   DATA[1204,17] := 1.0;
   DATA[1204,18] := 1.0;
   DATA[1204,19] := 1.0;
   DATA[1204,20] := 148.808;
   DATA[1204,21] := 154.2425;
   DATA[1204,22] := 1.716721;
   DATA[1204,23] := 841.2843;
   DATA[1204,24] := 2.0;
   DATA[1204,25] := 2.0;
   DATA[1204,26] := 7.87798;
   DATA[1204,27] := 143.5786;
   DATA[1204,28] := 263.0095;
   DATA[1204,29] := 12.07383;
   DATA[1204,30] := 1.725968;
   DATA[1204,31] := 1.298578;
   DATA[1204,32] := 0.7352687;
   DATA[1204,33] := 0.3083624;
   DATA[1204,34] := 2.0;
   DATA[1204,35] := 250.4166;
   DATA[1204,36] := 1.69801;
   DATA[1204,37] := 189.2944;
   DATA[1204,38] := 0.000128152;
   DATA[1204,39] := 1.0;
   DATA[1205,0] := 2.554527;
   DATA[1205,1] := 754.2025;
   DATA[1205,2] := 2.0;
   DATA[1205,3] := 1.0;
   DATA[1205,4] := 262.5288;
   DATA[1205,5] := 8.464369;
   DATA[1205,6] := 317.1494;
   DATA[1205,8] := 1.0;
   DATA[1205,9] := 1.0;
   DATA[1205,10] := 1.0;
   DATA[1205,11] := 2.010372;
   DATA[1205,12] := 0.000256221;
   DATA[1205,13] := 1011.079;
   DATA[1205,14] := 1.0;
   DATA[1205,15] := 1.0;
   DATA[1205,16] := 1.0;
   DATA[1205,17] := 1.0;
   DATA[1205,18] := 1.0;
   DATA[1205,19] := 1.0;
   DATA[1205,20] := 148.808;
   DATA[1205,21] := 154.2425;
   DATA[1205,22] := 1.717233;
   DATA[1205,23] := 840.8998;
   DATA[1205,24] := 2.0;
   DATA[1205,25] := 2.0;
   DATA[1205,26] := 7.87798;
   DATA[1205,27] := 143.5786;
   DATA[1205,28] := 263.0095;
   DATA[1205,29] := 12.26609;
   DATA[1205,30] := 1.725968;
   DATA[1205,31] := 1.301396;
   DATA[1205,32] := 0.7352687;
   DATA[1205,33] := 0.3083624;
   DATA[1205,34] := 2.0;
   DATA[1205,35] := 250.2724;
   DATA[1205,36] := 1.69801;
   DATA[1205,37] := 189.1342;
   DATA[1205,38] := 0.000128152;
   DATA[1205,39] := 1.0;
   DATA[1206,0] := 2.554527;
   DATA[1206,1] := 754.7128;
   DATA[1206,2] := 2.0;
   DATA[1206,3] := 1.0;
   DATA[1206,4] := 262.5288;
   DATA[1206,5] := 8.464369;
   DATA[1206,6] := 317.1494;
   DATA[1206,8] := 1.0;
   DATA[1206,9] := 1.0;
   DATA[1206,10] := 1.0;
   DATA[1206,11] := 2.010372;
   DATA[1206,12] := 0.000256221;
   DATA[1206,13] := 1010.919;
   DATA[1206,14] := 1.0;
   DATA[1206,15] := 1.0;
   DATA[1206,16] := 1.0;
   DATA[1206,17] := 1.0;
   DATA[1206,18] := 1.0;
   DATA[1206,19] := 1.0;
   DATA[1206,20] := 148.808;
   DATA[1206,21] := 154.2425;
   DATA[1206,22] := 1.717874;
   DATA[1206,23] := 840.7844;
   DATA[1206,24] := 2.0;
   DATA[1206,25] := 2.0;
   DATA[1206,26] := 7.87798;
   DATA[1206,27] := 143.5786;
   DATA[1206,28] := 263.0095;
   DATA[1206,29] := 12.26609;
   DATA[1206,30] := 1.72443;
   DATA[1206,31] := 1.291789;
   DATA[1206,32] := 0.7352687;
   DATA[1206,33] := 0.3083624;
   DATA[1206,34] := 2.0;
   DATA[1206,35] := 250.2724;
   DATA[1206,36] := 1.69801;
   DATA[1206,37] := 189.0381;
   DATA[1206,38] := 0.000128152;
   DATA[1206,39] := 1.0;
   DATA[1207,0] := 2.554527;
   DATA[1207,1] := 755.2623;
   DATA[1207,2] := 2.0;
   DATA[1207,3] := 1.0;
   DATA[1207,4] := 262.5288;
   DATA[1207,5] := 8.464369;
   DATA[1207,6] := 317.1494;
   DATA[1207,8] := 1.0;
   DATA[1207,9] := 1.0;
   DATA[1207,10] := 1.0;
   DATA[1207,11] := 2.010372;
   DATA[1207,12] := 0.000256221;
   DATA[1207,13] := 1011.159;
   DATA[1207,14] := 1.0;
   DATA[1207,15] := 1.0;
   DATA[1207,16] := 1.0;
   DATA[1207,17] := 1.0;
   DATA[1207,18] := 1.0;
   DATA[1207,19] := 1.0;
   DATA[1207,20] := 148.808;
   DATA[1207,21] := 154.2425;
   DATA[1207,22] := 1.717874;
   DATA[1207,23] := 840.2845;
   DATA[1207,24] := 2.0;
   DATA[1207,25] := 2.0;
   DATA[1207,26] := 7.87798;
   DATA[1207,27] := 143.4248;
   DATA[1207,28] := 263.0095;
   DATA[1207,29] := 12.26609;
   DATA[1207,30] := 1.722892;
   DATA[1207,31] := 1.284232;
   DATA[1207,32] := 0.7352687;
   DATA[1207,33] := 0.3083624;
   DATA[1207,34] := 2.0;
   DATA[1207,35] := 250.1442;
   DATA[1207,36] := 1.69801;
   DATA[1207,37] := 189.0381;
   DATA[1207,38] := 0.000128152;
   DATA[1207,39] := 1.0;
   DATA[1208,0] := 2.55805;
   DATA[1208,1] := 755.6941;
   DATA[1208,2] := 2.0;
   DATA[1208,3] := 1.0;
   DATA[1208,4] := 262.5288;
   DATA[1208,5] := 8.464369;
   DATA[1208,6] := 317.1494;
   DATA[1208,8] := 1.0;
   DATA[1208,9] := 1.0;
   DATA[1208,10] := 1.0;
   DATA[1208,11] := 2.010372;
   DATA[1208,12] := 0.000256221;
   DATA[1208,13] := 1010.718;
   DATA[1208,14] := 1.0;
   DATA[1208,15] := 1.0;
   DATA[1208,16] := 1.0;
   DATA[1208,17] := 1.0;
   DATA[1208,18] := 1.0;
   DATA[1208,19] := 1.0;
   DATA[1208,20] := 148.808;
   DATA[1208,21] := 154.2425;
   DATA[1208,22] := 1.717874;
   DATA[1208,23] := 840.2076;
   DATA[1208,24] := 2.0;
   DATA[1208,25] := 2.0;
   DATA[1208,26] := 7.87798;
   DATA[1208,27] := 143.4248;
   DATA[1208,28] := 263.0095;
   DATA[1208,29] := 12.03538;
   DATA[1208,30] := 1.722892;
   DATA[1208,31] := 1.272576;
   DATA[1208,32] := 0.7352687;
   DATA[1208,33] := 0.3083624;
   DATA[1208,34] := 2.0;
   DATA[1208,35] := 250.1442;
   DATA[1208,36] := 1.69801;
   DATA[1208,37] := 189.0381;
   DATA[1208,38] := 0.000128152;
   DATA[1208,39] := 1.0;
   DATA[1209,0] := 2.559651;
   DATA[1209,1] := 756.4791;
   DATA[1209,2] := 2.0;
   DATA[1209,3] := 1.0;
   DATA[1209,4] := 262.5288;
   DATA[1209,5] := 8.464369;
   DATA[1209,6] := 317.1494;
   DATA[1209,8] := 1.0;
   DATA[1209,9] := 1.0;
   DATA[1209,10] := 1.0;
   DATA[1209,11] := 2.010372;
   DATA[1209,12] := 0.000256221;
   DATA[1209,13] := 1010.919;
   DATA[1209,14] := 1.0;
   DATA[1209,15] := 1.0;
   DATA[1209,16] := 1.0;
   DATA[1209,17] := 1.0;
   DATA[1209,18] := 1.0;
   DATA[1209,19] := 1.0;
   DATA[1209,20] := 148.808;
   DATA[1209,21] := 154.1912;
   DATA[1209,22] := 1.715439;
   DATA[1209,23] := 839.9;
   DATA[1209,24] := 2.0;
   DATA[1209,25] := 2.0;
   DATA[1209,26] := 7.87798;
   DATA[1209,27] := 143.4248;
   DATA[1209,28] := 263.0095;
   DATA[1209,29] := 12.03538;
   DATA[1209,30] := 1.722892;
   DATA[1209,31] := 1.263738;
   DATA[1209,32] := 0.7352687;
   DATA[1209,33] := 0.3083624;
   DATA[1209,34] := 2.0;
   DATA[1209,35] := 250.1442;
   DATA[1209,36] := 1.69801;
   DATA[1209,37] := 189.0381;
   DATA[1209,38] := 0.000128152;
   DATA[1209,39] := 1.0;
   DATA[1210,0] := 2.550043;
   DATA[1210,1] := 756.9502;
   DATA[1210,2] := 2.0;
   DATA[1210,3] := 1.0;
   DATA[1210,4] := 262.5288;
   DATA[1210,5] := 8.464369;
   DATA[1210,6] := 317.1494;
   DATA[1210,8] := 1.0;
   DATA[1210,9] := 1.0;
   DATA[1210,10] := 1.0;
   DATA[1210,11] := 2.010372;
   DATA[1210,12] := 0.000256221;
   DATA[1210,13] := 1010.879;
   DATA[1210,14] := 1.0;
   DATA[1210,15] := 1.0;
   DATA[1210,16] := 1.0;
   DATA[1210,17] := 1.0;
   DATA[1210,18] := 1.0;
   DATA[1210,19] := 1.0;
   DATA[1210,20] := 148.808;
   DATA[1210,21] := 154.0374;
   DATA[1210,22] := 1.713261;
   DATA[1210,23] := 839.2848;
   DATA[1210,24] := 2.0;
   DATA[1210,25] := 2.0;
   DATA[1210,26] := 7.87798;
   DATA[1210,27] := 143.4248;
   DATA[1210,28] := 263.0095;
   DATA[1210,29] := 12.03538;
   DATA[1210,30] := 1.722892;
   DATA[1210,31] := 1.279237;
   DATA[1210,32] := 0.7352687;
   DATA[1210,33] := 0.3083624;
   DATA[1210,34] := 2.0;
   DATA[1210,35] := 250.1442;
   DATA[1210,36] := 1.69801;
   DATA[1210,37] := 189.0381;
   DATA[1210,38] := 0.000128152;
   DATA[1210,39] := 1.0;
   DATA[1211,0] := 2.550043;
   DATA[1211,1] := 757.853;
   DATA[1211,2] := 2.0;
   DATA[1211,3] := 1.0;
   DATA[1211,4] := 262.5288;
   DATA[1211,5] := 8.464369;
   DATA[1211,6] := 317.1494;
   DATA[1211,8] := 1.0;
   DATA[1211,9] := 1.0;
   DATA[1211,10] := 1.0;
   DATA[1211,11] := 2.010372;
   DATA[1211,12] := 0.000256221;
   DATA[1211,13] := 1010.879;
   DATA[1211,14] := 1.0;
   DATA[1211,15] := 1.0;
   DATA[1211,16] := 1.0;
   DATA[1211,17] := 1.0;
   DATA[1211,18] := 1.0;
   DATA[1211,19] := 1.0;
   DATA[1211,20] := 148.808;
   DATA[1211,21] := 153.8836;
   DATA[1211,22] := 1.711723;
   DATA[1211,23] := 839.3232;
   DATA[1211,24] := 2.0;
   DATA[1211,25] := 2.0;
   DATA[1211,26] := 7.87798;
   DATA[1211,27] := 143.4248;
   DATA[1211,28] := 263.0095;
   DATA[1211,29] := 12.03538;
   DATA[1211,30] := 1.722379;
   DATA[1211,31] := 1.289484;
   DATA[1211,32] := 0.7352687;
   DATA[1211,33] := 0.3083624;
   DATA[1211,34] := 2.0;
   DATA[1211,35] := 250.1442;
   DATA[1211,36] := 1.69801;
   DATA[1211,37] := 189.0381;
   DATA[1211,38] := 0.000128152;
   DATA[1211,39] := 1.0;
   DATA[1212,0] := 2.552285;
   DATA[1212,1] := 758.0885;
   DATA[1212,2] := 2.0;
   DATA[1212,3] := 1.0;
   DATA[1212,4] := 262.5288;
   DATA[1212,5] := 8.464369;
   DATA[1212,6] := 317.1494;
   DATA[1212,8] := 1.0;
   DATA[1212,9] := 1.0;
   DATA[1212,10] := 1.0;
   DATA[1212,11] := 2.010372;
   DATA[1212,12] := 0.000256221;
   DATA[1212,13] := 1010.718;
   DATA[1212,14] := 1.0;
   DATA[1212,15] := 1.0;
   DATA[1212,16] := 1.0;
   DATA[1212,17] := 1.0;
   DATA[1212,18] := 1.0;
   DATA[1212,19] := 1.0;
   DATA[1212,20] := 148.808;
   DATA[1212,21] := 153.8836;
   DATA[1212,22] := 1.711082;
   DATA[1212,23] := 838.8618;
   DATA[1212,24] := 2.0;
   DATA[1212,25] := 2.0;
   DATA[1212,26] := 7.87798;
   DATA[1212,27] := 143.4248;
   DATA[1212,28] := 263.0095;
   DATA[1212,29] := 12.03538;
   DATA[1212,30] := 1.722379;
   DATA[1212,31] := 1.299731;
   DATA[1212,32] := 0.7352687;
   DATA[1212,33] := 0.3083624;
   DATA[1212,34] := 2.0;
   DATA[1212,35] := 250.3525;
   DATA[1212,36] := 1.69801;
   DATA[1212,37] := 189.0381;
   DATA[1212,38] := 0.000128152;
   DATA[1212,39] := 1.0;
   DATA[1213,0] := 2.554847;
   DATA[1213,1] := 758.7166;
   DATA[1213,2] := 2.0;
   DATA[1213,3] := 1.0;
   DATA[1213,4] := 262.5288;
   DATA[1213,5] := 8.464369;
   DATA[1213,6] := 317.1494;
   DATA[1213,8] := 1.0;
   DATA[1213,9] := 1.0;
   DATA[1213,10] := 1.0;
   DATA[1213,11] := 2.010372;
   DATA[1213,12] := 0.000256221;
   DATA[1213,13] := 1010.478;
   DATA[1213,14] := 1.0;
   DATA[1213,15] := 1.0;
   DATA[1213,16] := 1.0;
   DATA[1213,17] := 1.0;
   DATA[1213,18] := 1.0;
   DATA[1213,19] := 1.0;
   DATA[1213,20] := 148.808;
   DATA[1213,21] := 153.8836;
   DATA[1213,22] := 1.711082;
   DATA[1213,23] := 838.5542;
   DATA[1213,24] := 2.0;
   DATA[1213,25] := 2.0;
   DATA[1213,26] := 7.87798;
   DATA[1213,27] := 143.4248;
   DATA[1213,28] := 263.0095;
   DATA[1213,29] := 12.03538;
   DATA[1213,30] := 1.722379;
   DATA[1213,31] := 1.30114;
   DATA[1213,32] := 0.7352687;
   DATA[1213,33] := 0.3083624;
   DATA[1213,34] := 2.0;
   DATA[1213,35] := 250.3525;
   DATA[1213,36] := 1.69801;
   DATA[1213,37] := 189.0541;
   DATA[1213,38] := 0.000128152;
   DATA[1213,39] := 1.0;
   DATA[1214,0] := 2.556129;
   DATA[1214,1] := 759.4231;
   DATA[1214,2] := 2.0;
   DATA[1214,3] := 1.0;
   DATA[1214,4] := 262.5288;
   DATA[1214,5] := 8.464369;
   DATA[1214,6] := 317.1494;
   DATA[1214,8] := 1.0;
   DATA[1214,9] := 1.0;
   DATA[1214,10] := 1.0;
   DATA[1214,11] := 2.010372;
   DATA[1214,12] := 0.000256221;
   DATA[1214,13] := 1010.718;
   DATA[1214,14] := 1.0;
   DATA[1214,15] := 1.0;
   DATA[1214,16] := 1.0;
   DATA[1214,17] := 1.0;
   DATA[1214,18] := 1.0;
   DATA[1214,19] := 1.0;
   DATA[1214,20] := 148.808;
   DATA[1214,21] := 154.0118;
   DATA[1214,22] := 1.712363;
   DATA[1214,23] := 838.0543;
   DATA[1214,24] := 2.0;
   DATA[1214,25] := 2.0;
   DATA[1214,26] := 7.87798;
   DATA[1214,27] := 143.3222;
   DATA[1214,28] := 263.0095;
   DATA[1214,29] := 12.03538;
   DATA[1214,30] := 1.725583;
   DATA[1214,31] := 1.291789;
   DATA[1214,32] := 0.7352687;
   DATA[1214,33] := 0.3074656;
   DATA[1214,34] := 2.0;
   DATA[1214,35] := 250.3525;
   DATA[1214,36] := 1.69801;
   DATA[1214,37] := 189.2143;
   DATA[1214,38] := 0.000128152;
   DATA[1214,39] := 1.0;
   DATA[1215,0] := 2.556129;
   DATA[1215,1] := 760.4044;
   DATA[1215,2] := 2.0;
   DATA[1215,3] := 1.0;
   DATA[1215,4] := 262.5288;
   DATA[1215,5] := 8.464369;
   DATA[1215,6] := 317.1494;
   DATA[1215,8] := 1.0;
   DATA[1215,9] := 1.0;
   DATA[1215,10] := 1.0;
   DATA[1215,11] := 2.010372;
   DATA[1215,12] := 0.000256221;
   DATA[1215,13] := 1010.558;
   DATA[1215,14] := 1.0;
   DATA[1215,15] := 1.0;
   DATA[1215,16] := 1.0;
   DATA[1215,17] := 1.0;
   DATA[1215,18] := 1.0;
   DATA[1215,19] := 1.0;
   DATA[1215,20] := 148.808;
   DATA[1215,21] := 154.0118;
   DATA[1215,22] := 1.715567;
   DATA[1215,23] := 837.7852;
   DATA[1215,24] := 2.0;
   DATA[1215,25] := 2.0;
   DATA[1215,26] := 7.87798;
   DATA[1215,27] := 143.2966;
   DATA[1215,28] := 263.0095;
   DATA[1215,29] := 12.03538;
   DATA[1215,30] := 1.72725;
   DATA[1215,31] := 1.282183;
   DATA[1215,32] := 0.7352687;
   DATA[1215,33] := 0.3068891;
   DATA[1215,34] := 2.0;
   DATA[1215,35] := 250.4967;
   DATA[1215,36] := 1.69801;
   DATA[1215,37] := 189.2143;
   DATA[1215,38] := 0.000128152;
   DATA[1215,39] := 1.0;
   DATA[1216,0] := 2.553566;
   DATA[1216,1] := 760.9932;
   DATA[1216,2] := 2.0;
   DATA[1216,3] := 1.0;
   DATA[1216,4] := 262.5288;
   DATA[1216,5] := 8.464369;
   DATA[1216,6] := 317.1494;
   DATA[1216,8] := 1.0;
   DATA[1216,9] := 1.0;
   DATA[1216,10] := 1.0;
   DATA[1216,11] := 2.010372;
   DATA[1216,12] := 0.000256221;
   DATA[1216,13] := 1010.959;
   DATA[1216,14] := 1.0;
   DATA[1216,15] := 1.0;
   DATA[1216,16] := 1.0;
   DATA[1216,17] := 1.0;
   DATA[1216,18] := 1.0;
   DATA[1216,19] := 1.0;
   DATA[1216,20] := 148.808;
   DATA[1216,21] := 154.0118;
   DATA[1216,22] := 1.716721;
   DATA[1216,23] := 837.2853;
   DATA[1216,24] := 2.0;
   DATA[1216,25] := 2.0;
   DATA[1216,26] := 7.87798;
   DATA[1216,27] := 143.2966;
   DATA[1216,28] := 263.0095;
   DATA[1216,29] := 12.03538;
   DATA[1216,30] := 1.727378;
   DATA[1216,31] := 1.273857;
   DATA[1216,32] := 0.7352687;
   DATA[1216,33] := 0.3068891;
   DATA[1216,34] := 2.0;
   DATA[1216,35] := 250.4967;
   DATA[1216,36] := 1.69801;
   DATA[1216,37] := 189.2624;
   DATA[1216,38] := 0.000128152;
   DATA[1216,39] := 1.0;
   DATA[1217,0] := 2.550684;
   DATA[1217,1] := 761.3465;
   DATA[1217,2] := 2.0;
   DATA[1217,3] := 1.0;
   DATA[1217,4] := 262.5288;
   DATA[1217,5] := 8.464369;
   DATA[1217,6] := 317.2263;
   DATA[1217,8] := 1.0;
   DATA[1217,9] := 1.0;
   DATA[1217,10] := 1.0;
   DATA[1217,11] := 2.010372;
   DATA[1217,12] := 0.000256221;
   DATA[1217,13] := 1010.758;
   DATA[1217,14] := 1.0;
   DATA[1217,15] := 1.0;
   DATA[1217,16] := 1.0;
   DATA[1217,17] := 1.0;
   DATA[1217,18] := 1.0;
   DATA[1217,19] := 1.0;
   DATA[1217,20] := 148.808;
   DATA[1217,21] := 154.0118;
   DATA[1217,22] := 1.716849;
   DATA[1217,23] := 837.516;
   DATA[1217,24] := 2.0;
   DATA[1217,25] := 2.0;
   DATA[1217,26] := 7.87798;
   DATA[1217,27] := 143.2966;
   DATA[1217,28] := 263.0095;
   DATA[1217,29] := 12.03538;
   DATA[1217,30] := 1.727378;
   DATA[1217,31] := 1.287947;
   DATA[1217,32] := 0.7352687;
   DATA[1217,33] := 0.3068891;
   DATA[1217,34] := 2.0;
   DATA[1217,35] := 250.5127;
   DATA[1217,36] := 1.69801;
   DATA[1217,37] := 189.2624;
   DATA[1217,38] := 0.000128152;
   DATA[1217,39] := 1.0;
   DATA[1218,0] := 2.550684;
   DATA[1218,1] := 762.524;
   DATA[1218,2] := 2.0;
   DATA[1218,3] := 1.0;
   DATA[1218,4] := 262.5288;
   DATA[1218,5] := 8.464369;
   DATA[1218,6] := 317.2263;
   DATA[1218,8] := 1.0;
   DATA[1218,9] := 1.0;
   DATA[1218,10] := 1.0;
   DATA[1218,11] := 2.010372;
   DATA[1218,12] := 0.000256221;
   DATA[1218,13] := 1010.718;
   DATA[1218,14] := 1.0;
   DATA[1218,15] := 1.0;
   DATA[1218,16] := 1.0;
   DATA[1218,17] := 1.0;
   DATA[1218,18] := 1.0;
   DATA[1218,19] := 1.0;
   DATA[1218,20] := 148.808;
   DATA[1218,21] := 154.0118;
   DATA[1218,22] := 1.716849;
   DATA[1218,23] := 837.17;
   DATA[1218,24] := 2.0;
   DATA[1218,25] := 2.0;
   DATA[1218,26] := 7.87798;
   DATA[1218,27] := 143.2966;
   DATA[1218,28] := 263.0095;
   DATA[1218,29] := 12.03538;
   DATA[1218,30] := 1.727378;
   DATA[1218,31] := 1.3005;
   DATA[1218,32] := 0.7352687;
   DATA[1218,33] := 0.3066329;
   DATA[1218,34] := 2.0;
   DATA[1218,35] := 250.5127;
   DATA[1218,36] := 1.69801;
   DATA[1218,37] := 189.3745;
   DATA[1218,38] := 0.000128152;
   DATA[1218,39] := 1.0;
   DATA[1219,0] := 2.551324;
   DATA[1219,1] := 762.8381;
   DATA[1219,2] := 2.0;
   DATA[1219,3] := 1.0;
   DATA[1219,4] := 262.5288;
   DATA[1219,5] := 8.464369;
   DATA[1219,6] := 317.2263;
   DATA[1219,8] := 1.0;
   DATA[1219,9] := 1.0;
   DATA[1219,10] := 1.0;
   DATA[1219,11] := 2.010372;
   DATA[1219,12] := 0.000256221;
   DATA[1219,13] := 1010.879;
   DATA[1219,14] := 1.0;
   DATA[1219,15] := 1.0;
   DATA[1219,16] := 1.0;
   DATA[1219,17] := 1.0;
   DATA[1219,18] := 1.0;
   DATA[1219,19] := 1.0;
   DATA[1219,20] := 148.808;
   DATA[1219,21] := 154.0118;
   DATA[1219,22] := 1.717233;
   DATA[1219,23] := 836.6317;
   DATA[1219,24] := 2.0;
   DATA[1219,25] := 2.0;
   DATA[1219,26] := 7.87798;
   DATA[1219,27] := 143.2966;
   DATA[1219,28] := 263.0095;
   DATA[1219,29] := 12.03538;
   DATA[1219,30] := 1.728531;
   DATA[1219,31] := 1.302037;
   DATA[1219,32] := 0.7352687;
   DATA[1219,33] := 0.3066329;
   DATA[1219,34] := 2.0;
   DATA[1219,35] := 250.5127;
   DATA[1219,36] := 1.69801;
   DATA[1219,37] := 189.3745;
   DATA[1219,38] := 0.000128152;
   DATA[1219,39] := 1.0;
   DATA[1220,0] := 2.551324;
   DATA[1220,1] := 763.5839;
   DATA[1220,2] := 2.0;
   DATA[1220,3] := 1.0;
   DATA[1220,4] := 262.5288;
   DATA[1220,5] := 8.464369;
   DATA[1220,6] := 317.2263;
   DATA[1220,8] := 1.0;
   DATA[1220,9] := 1.0;
   DATA[1220,10] := 1.0;
   DATA[1220,11] := 2.010372;
   DATA[1220,12] := 0.000256221;
   DATA[1220,13] := 1010.839;
   DATA[1220,14] := 1.0;
   DATA[1220,15] := 1.0;
   DATA[1220,16] := 1.0;
   DATA[1220,17] := 1.0;
   DATA[1220,18] := 1.0;
   DATA[1220,19] := 1.0;
   DATA[1220,20] := 148.808;
   DATA[1220,21] := 154.0118;
   DATA[1220,22] := 1.717489;
   DATA[1220,23] := 836.2471;
   DATA[1220,24] := 2.0;
   DATA[1220,25] := 2.0;
   DATA[1220,26] := 7.87798;
   DATA[1220,27] := 143.2966;
   DATA[1220,28] := 263.0095;
   DATA[1220,29] := 12.26609;
   DATA[1220,30] := 1.728531;
   DATA[1220,31] := 1.302037;
   DATA[1220,32] := 0.7352687;
   DATA[1220,33] := 0.3066329;
   DATA[1220,34] := 2.0;
   DATA[1220,35] := 250.5127;
   DATA[1220,36] := 1.69801;
   DATA[1220,37] := 189.3745;
   DATA[1220,38] := 0.000128152;
   DATA[1220,39] := 1.0;
   DATA[1221,0] := 2.543958;
   DATA[1221,1] := 764.212;
   DATA[1221,2] := 2.0;
   DATA[1221,3] := 1.0;
   DATA[1221,4] := 262.5288;
   DATA[1221,5] := 8.464369;
   DATA[1221,6] := 317.2263;
   DATA[1221,8] := 1.0;
   DATA[1221,9] := 1.0;
   DATA[1221,10] := 1.0;
   DATA[1221,11] := 2.010372;
   DATA[1221,12] := 0.000256221;
   DATA[1221,13] := 1010.839;
   DATA[1221,14] := 1.0;
   DATA[1221,15] := 1.0;
   DATA[1221,16] := 1.0;
   DATA[1221,17] := 1.0;
   DATA[1221,18] := 1.0;
   DATA[1221,19] := 1.0;
   DATA[1221,20] := 148.808;
   DATA[1221,21] := 154.2425;
   DATA[1221,22] := 1.717489;
   DATA[1221,23] := 835.978;
   DATA[1221,24] := 2.0;
   DATA[1221,25] := 2.0;
   DATA[1221,26] := 7.87798;
   DATA[1221,27] := 143.2966;
   DATA[1221,28] := 263.0095;
   DATA[1221,29] := 12.26609;
   DATA[1221,30] := 1.728531;
   DATA[1221,31] := 1.30178;
   DATA[1221,32] := 0.7352687;
   DATA[1221,33] := 0.3066329;
   DATA[1221,34] := 2.0;
   DATA[1221,35] := 250.5127;
   DATA[1221,36] := 1.69801;
   DATA[1221,37] := 189.3745;
   DATA[1221,38] := 0.000128152;
   DATA[1221,39] := 1.0;
   DATA[1222,0] := 2.543638;
   DATA[1222,1] := 765.154;
   DATA[1222,2] := 2.0;
   DATA[1222,3] := 1.0;
   DATA[1222,4] := 262.5288;
   DATA[1222,5] := 8.464369;
   DATA[1222,6] := 317.2263;
   DATA[1222,8] := 1.0;
   DATA[1222,9] := 1.0;
   DATA[1222,10] := 1.0;
   DATA[1222,11] := 2.010372;
   DATA[1222,12] := 0.000256221;
   DATA[1222,13] := 1010.678;
   DATA[1222,14] := 1.0;
   DATA[1222,15] := 1.0;
   DATA[1222,16] := 1.0;
   DATA[1222,17] := 1.0;
   DATA[1222,18] := 1.0;
   DATA[1222,19] := 1.0;
   DATA[1222,20] := 148.808;
   DATA[1222,21] := 154.2425;
   DATA[1222,22] := 1.71467;
   DATA[1222,23] := 835.3627;
   DATA[1222,24] := 2.0;
   DATA[1222,25] := 2.0;
   DATA[1222,26] := 7.87798;
   DATA[1222,27] := 143.2966;
   DATA[1222,28] := 263.0095;
   DATA[1222,29] := 11.95847;
   DATA[1222,30] := 1.728531;
   DATA[1222,31] := 1.291405;
   DATA[1222,32] := 0.7352687;
   DATA[1222,33] := 0.3066329;
   DATA[1222,34] := 2.0;
   DATA[1222,35] := 250.5127;
   DATA[1222,36] := 1.69801;
   DATA[1222,37] := 189.3745;
   DATA[1222,38] := 0.000128152;
   DATA[1222,39] := 1.0;
   DATA[1223,0] := 2.547161;
   DATA[1223,1] := 765.154;
   DATA[1223,2] := 2.0;
   DATA[1223,3] := 1.0;
   DATA[1223,4] := 262.5288;
   DATA[1223,5] := 8.464369;
   DATA[1223,6] := 317.2263;
   DATA[1223,8] := 1.0;
   DATA[1223,9] := 1.0;
   DATA[1223,10] := 1.0;
   DATA[1223,11] := 2.010372;
   DATA[1223,12] := 0.000256221;
   DATA[1223,13] := 1010.678;
   DATA[1223,14] := 1.0;
   DATA[1223,15] := 1.0;
   DATA[1223,16] := 1.0;
   DATA[1223,17] := 1.0;
   DATA[1223,18] := 1.0;
   DATA[1223,19] := 1.0;
   DATA[1223,20] := 148.808;
   DATA[1223,21] := 154.2425;
   DATA[1223,22] := 1.71262;
   DATA[1223,23] := 834.8244;
   DATA[1223,24] := 2.0;
   DATA[1223,25] := 2.0;
   DATA[1223,26] := 7.87798;
   DATA[1223,27] := 143.2966;
   DATA[1223,28] := 263.1056;
   DATA[1223,29] := 11.95847;
   DATA[1223,30] := 1.726609;
   DATA[1223,31] := 1.291405;
   DATA[1223,32] := 0.7352687;
   DATA[1223,33] := 0.3066329;
   DATA[1223,34] := 2.0;
   DATA[1223,35] := 250.5127;
   DATA[1223,36] := 1.69801;
   DATA[1223,37] := 189.3745;
   DATA[1223,38] := 0.000128152;
   DATA[1223,39] := 1.0;
   DATA[1224,0] := 2.556449;
   DATA[1224,1] := 765.7036;
   DATA[1224,2] := 2.0;
   DATA[1224,3] := 1.0;
   DATA[1224,4] := 262.5288;
   DATA[1224,5] := 8.464369;
   DATA[1224,6] := 317.2263;
   DATA[1224,8] := 1.0;
   DATA[1224,9] := 1.0;
   DATA[1224,10] := 1.0;
   DATA[1224,11] := 2.010372;
   DATA[1224,12] := 0.000256221;
   DATA[1224,13] := 1011.039;
   DATA[1224,14] := 1.0;
   DATA[1224,15] := 1.0;
   DATA[1224,16] := 1.0;
   DATA[1224,17] := 1.0;
   DATA[1224,18] := 1.0;
   DATA[1224,19] := 1.0;
   DATA[1224,20] := 148.808;
   DATA[1224,21] := 154.1143;
   DATA[1224,22] := 1.71262;
   DATA[1224,23] := 834.5937;
   DATA[1224,24] := 2.0;
   DATA[1224,25] := 2.0;
   DATA[1224,26] := 7.87798;
   DATA[1224,27] := 143.2966;
   DATA[1224,28] := 263.1056;
   DATA[1224,29] := 11.95847;
   DATA[1224,30] := 1.726609;
   DATA[1224,31] := 1.298578;
   DATA[1224,32] := 0.7352687;
   DATA[1224,33] := 0.3066329;
   DATA[1224,34] := 2.0;
   DATA[1224,35] := 250.5127;
   DATA[1224,36] := 1.69801;
   DATA[1224,37] := 189.3745;
   DATA[1224,38] := 0.000128152;
   DATA[1224,39] := 1.0;
   DATA[1225,0] := 2.558691;
   DATA[1225,1] := 766.3708;
   DATA[1225,2] := 2.0;
   DATA[1225,3] := 1.0;
   DATA[1225,4] := 262.5288;
   DATA[1225,5] := 8.464369;
   DATA[1225,6] := 317.4058;
   DATA[1225,8] := 1.0;
   DATA[1225,9] := 1.0;
   DATA[1225,10] := 1.0;
   DATA[1225,11] := 2.010372;
   DATA[1225,12] := 0.000256221;
   DATA[1225,13] := 1011.279;
   DATA[1225,14] := 1.0;
   DATA[1225,15] := 1.0;
   DATA[1225,16] := 1.0;
   DATA[1225,17] := 1.0;
   DATA[1225,18] := 1.0;
   DATA[1225,19] := 1.0;
   DATA[1225,20] := 148.808;
   DATA[1225,21] := 154.1143;
   DATA[1225,22] := 1.711595;
   DATA[1225,23] := 834.0554;
   DATA[1225,24] := 2.0;
   DATA[1225,25] := 2.0;
   DATA[1225,26] := 7.87798;
   DATA[1225,27] := 143.2966;
   DATA[1225,28] := 263.1056;
   DATA[1225,29] := 11.95847;
   DATA[1225,30] := 1.726609;
   DATA[1225,31] := 1.283848;
   DATA[1225,32] := 0.7352687;
   DATA[1225,33] := 0.3066329;
   DATA[1225,34] := 2.0;
   DATA[1225,35] := 250.5127;
   DATA[1225,36] := 1.69801;
   DATA[1225,37] := 189.3745;
   DATA[1225,38] := 0.000128152;
   DATA[1225,39] := 1.0;
   DATA[1226,0] := 2.558691;
   DATA[1226,1] := 766.8419;
   DATA[1226,2] := 2.0;
   DATA[1226,3] := 1.0;
   DATA[1226,4] := 262.5288;
   DATA[1226,5] := 8.464369;
   DATA[1226,6] := 317.4058;
   DATA[1226,8] := 1.0;
   DATA[1226,9] := 1.0;
   DATA[1226,10] := 1.0;
   DATA[1226,11] := 2.010372;
   DATA[1226,12] := 0.000256221;
   DATA[1226,13] := 1011.159;
   DATA[1226,14] := 1.0;
   DATA[1226,15] := 1.0;
   DATA[1226,16] := 1.0;
   DATA[1226,17] := 1.0;
   DATA[1226,18] := 1.0;
   DATA[1226,19] := 1.0;
   DATA[1226,20] := 148.808;
   DATA[1226,21] := 154.1143;
   DATA[1226,22] := 1.711595;
   DATA[1226,23] := 833.9016;
   DATA[1226,24] := 2.0;
   DATA[1226,25] := 2.0;
   DATA[1226,26] := 7.87798;
   DATA[1226,27] := 143.2966;
   DATA[1226,28] := 263.1056;
   DATA[1226,29] := 11.95847;
   DATA[1226,30] := 1.726609;
   DATA[1226,31] := 1.281798;
   DATA[1226,32] := 0.7352687;
   DATA[1226,33] := 0.3066329;
   DATA[1226,34] := 2.0;
   DATA[1226,35] := 250.5127;
   DATA[1226,36] := 1.69801;
   DATA[1226,37] := 189.2143;
   DATA[1226,38] := 0.000128152;
   DATA[1226,39] := 1.0;
   DATA[1227,0] := 2.558691;
   DATA[1227,1] := 767.0381;
   DATA[1227,2] := 2.0;
   DATA[1227,3] := 1.0;
   DATA[1227,4] := 262.5288;
   DATA[1227,5] := 8.464369;
   DATA[1227,6] := 317.4058;
   DATA[1227,8] := 1.0;
   DATA[1227,9] := 1.0;
   DATA[1227,10] := 1.0;
   DATA[1227,11] := 2.010372;
   DATA[1227,12] := 0.000256221;
   DATA[1227,13] := 1011.119;
   DATA[1227,14] := 1.0;
   DATA[1227,15] := 1.0;
   DATA[1227,16] := 1.0;
   DATA[1227,17] := 1.0;
   DATA[1227,18] := 1.0;
   DATA[1227,19] := 1.0;
   DATA[1227,20] := 148.808;
   DATA[1227,21] := 154.1143;
   DATA[1227,22] := 1.712748;
   DATA[1227,23] := 833.3632;
   DATA[1227,24] := 2.0;
   DATA[1227,25] := 2.0;
   DATA[1227,26] := 7.87798;
   DATA[1227,27] := 143.2966;
   DATA[1227,28] := 263.1056;
   DATA[1227,29] := 11.95847;
   DATA[1227,30] := 1.726609;
   DATA[1227,31] := 1.281798;
   DATA[1227,32] := 0.7352687;
   DATA[1227,33] := 0.3083624;
   DATA[1227,34] := 2.0;
   DATA[1227,35] := 250.5127;
   DATA[1227,36] := 1.681991;
   DATA[1227,37] := 189.1983;
   DATA[1227,38] := 0.000128152;
   DATA[1227,39] := 1.0;
   DATA[1228,0] := 2.558691;
   DATA[1228,1] := 767.5092;
   DATA[1228,2] := 2.0;
   DATA[1228,3] := 1.0;
   DATA[1228,4] := 262.5288;
   DATA[1228,5] := 8.464369;
   DATA[1228,6] := 317.4058;
   DATA[1228,8] := 1.0;
   DATA[1228,9] := 1.0;
   DATA[1228,10] := 1.0;
   DATA[1228,11] := 2.010372;
   DATA[1228,12] := 0.000256221;
   DATA[1228,13] := 1011.039;
   DATA[1228,14] := 1.0;
   DATA[1228,15] := 1.0;
   DATA[1228,16] := 1.0;
   DATA[1228,17] := 1.0;
   DATA[1228,18] := 1.0;
   DATA[1228,19] := 1.0;
   DATA[1228,20] := 148.808;
   DATA[1228,21] := 154.1143;
   DATA[1228,22] := 1.713261;
   DATA[1228,23] := 832.9402;
   DATA[1228,24] := 2.0;
   DATA[1228,25] := 2.0;
   DATA[1228,26] := 7.87798;
   DATA[1228,27] := 143.2966;
   DATA[1228,28] := 263.1056;
   DATA[1228,29] := 11.95847;
   DATA[1228,30] := 1.725968;
   DATA[1228,31] := 1.291405;
   DATA[1228,32] := 0.7352687;
   DATA[1228,33] := 0.3083624;
   DATA[1228,34] := 2.0;
   DATA[1228,35] := 250.5127;
   DATA[1228,36] := 1.681991;
   DATA[1228,37] := 189.1983;
   DATA[1228,38] := 0.000128152;
   DATA[1228,39] := 1.0;
   DATA[1229,0] := 2.558691;
   DATA[1229,1] := 768.0195;
   DATA[1229,2] := 2.0;
   DATA[1229,3] := 1.0;
   DATA[1229,4] := 262.5288;
   DATA[1229,5] := 8.464369;
   DATA[1229,6] := 317.4058;
   DATA[1229,8] := 1.0;
   DATA[1229,9] := 1.0;
   DATA[1229,10] := 1.0;
   DATA[1229,11] := 2.010372;
   DATA[1229,12] := 0.000256221;
   DATA[1229,13] := 1010.839;
   DATA[1229,14] := 1.0;
   DATA[1229,15] := 1.0;
   DATA[1229,16] := 1.0;
   DATA[1229,17] := 1.0;
   DATA[1229,18] := 1.0;
   DATA[1229,19] := 1.0;
   DATA[1229,20] := 148.808;
   DATA[1229,21] := 154.1143;
   DATA[1229,22] := 1.713261;
   DATA[1229,23] := 832.4789;
   DATA[1229,24] := 2.0;
   DATA[1229,25] := 2.0;
   DATA[1229,26] := 7.87798;
   DATA[1229,27] := 143.2966;
   DATA[1229,28] := 263.1056;
   DATA[1229,29] := 11.95847;
   DATA[1229,30] := 1.725968;
   DATA[1229,31] := 1.300243;
   DATA[1229,32] := 0.7352687;
   DATA[1229,33] := 0.3083624;
   DATA[1229,34] := 2.0;
   DATA[1229,35] := 250.5127;
   DATA[1229,36] := 1.681991;
   DATA[1229,37] := 189.1983;
   DATA[1229,38] := 0.000128152;
   DATA[1229,39] := 1.0;
   DATA[1230,0] := 2.547161;
   DATA[1230,1] := 768.726;
   DATA[1230,2] := 2.0;
   DATA[1230,3] := 1.0;
   DATA[1230,4] := 262.5288;
   DATA[1230,5] := 8.464369;
   DATA[1230,6] := 317.4058;
   DATA[1230,8] := 1.0;
   DATA[1230,9] := 1.0;
   DATA[1230,10] := 1.0;
   DATA[1230,11] := 2.010372;
   DATA[1230,12] := 0.000256221;
   DATA[1230,13] := 1010.638;
   DATA[1230,14] := 1.0;
   DATA[1230,15] := 1.0;
   DATA[1230,16] := 1.0;
   DATA[1230,17] := 1.0;
   DATA[1230,18] := 1.0;
   DATA[1230,19] := 1.0;
   DATA[1230,20] := 148.808;
   DATA[1230,21] := 154.1143;
   DATA[1230,22] := 1.712235;
   DATA[1230,23] := 831.9406;
   DATA[1230,24] := 2.0;
   DATA[1230,25] := 2.0;
   DATA[1230,26] := 7.87798;
   DATA[1230,27] := 143.2966;
   DATA[1230,28] := 263.1056;
   DATA[1230,29] := 12.15073;
   DATA[1230,30] := 1.725968;
   DATA[1230,31] := 1.301396;
   DATA[1230,32] := 0.7352687;
   DATA[1230,33] := 0.3083624;
   DATA[1230,34] := 2.0;
   DATA[1230,35] := 250.1122;
   DATA[1230,36] := 1.681991;
   DATA[1230,37] := 189.0381;
   DATA[1230,38] := 0.000128152;
   DATA[1230,39] := 1.0;
   DATA[1231,0] := 2.540115;
   DATA[1231,1] := 769.1185;
   DATA[1231,2] := 2.0;
   DATA[1231,3] := 1.0;
   DATA[1231,4] := 262.5288;
   DATA[1231,5] := 8.464369;
   DATA[1231,6] := 317.4058;
   DATA[1231,8] := 1.0;
   DATA[1231,9] := 1.0;
   DATA[1231,10] := 1.0;
   DATA[1231,11] := 2.010372;
   DATA[1231,12] := 0.000256221;
   DATA[1231,13] := 1010.879;
   DATA[1231,14] := 1.0;
   DATA[1231,15] := 1.0;
   DATA[1231,16] := 1.0;
   DATA[1231,17] := 1.0;
   DATA[1231,18] := 1.0;
   DATA[1231,19] := 1.0;
   DATA[1231,20] := 148.808;
   DATA[1231,21] := 154.1143;
   DATA[1231,22] := 1.710826;
   DATA[1231,23] := 832.0944;
   DATA[1231,24] := 2.0;
   DATA[1231,25] := 2.0;
   DATA[1231,26] := 7.87798;
   DATA[1231,27] := 143.2966;
   DATA[1231,28] := 263.1056;
   DATA[1231,29] := 12.15073;
   DATA[1231,30] := 1.72507;
   DATA[1231,31] := 1.282311;
   DATA[1231,32] := 0.7352687;
   DATA[1231,33] := 0.3083624;
   DATA[1231,34] := 2.0;
   DATA[1231,35] := 250.1122;
   DATA[1231,36] := 1.681991;
   DATA[1231,37] := 189.0381;
   DATA[1231,38] := 0.000128152;
   DATA[1231,39] := 1.0;
   DATA[1232,0] := 2.532748;
   DATA[1232,1] := 769.2756;
   DATA[1232,2] := 2.0;
   DATA[1232,3] := 1.0;
   DATA[1232,4] := 262.5288;
   DATA[1232,5] := 8.464369;
   DATA[1232,6] := 317.4058;
   DATA[1232,8] := 1.0;
   DATA[1232,9] := 1.0;
   DATA[1232,10] := 1.0;
   DATA[1232,11] := 2.010372;
   DATA[1232,12] := 0.000256221;
   DATA[1232,13] := 1011.039;
   DATA[1232,14] := 1.0;
   DATA[1232,15] := 1.0;
   DATA[1232,16] := 1.0;
   DATA[1232,17] := 1.0;
   DATA[1232,18] := 1.0;
   DATA[1232,19] := 1.0;
   DATA[1232,20] := 148.808;
   DATA[1232,21] := 154.1143;
   DATA[1232,22] := 1.710826;
   DATA[1232,23] := 831.7098;
   DATA[1232,24] := 2.0;
   DATA[1232,25] := 2.0;
   DATA[1232,26] := 7.87798;
   DATA[1232,27] := 143.2966;
   DATA[1232,28] := 263.1056;
   DATA[1232,29] := 12.15073;
   DATA[1232,30] := 1.723404;
   DATA[1232,31] := 1.275778;
   DATA[1232,32] := 0.7352687;
   DATA[1232,33] := 0.3083624;
   DATA[1232,34] := 2.0;
   DATA[1232,35] := 250.1122;
   DATA[1232,36] := 1.681991;
   DATA[1232,37] := 188.8138;
   DATA[1232,38] := 0.000128152;
   DATA[1232,39] := 1.0;
   DATA[1233,0] := 2.527624;
   DATA[1233,1] := 769.8643;
   DATA[1233,2] := 2.0;
   DATA[1233,3] := 1.0;
   DATA[1233,4] := 262.5288;
   DATA[1233,5] := 8.464048;
   DATA[1233,6] := 317.4058;
   DATA[1233,8] := 1.0;
   DATA[1233,9] := 1.0;
   DATA[1233,10] := 1.0;
   DATA[1233,11] := 2.010372;
   DATA[1233,12] := 0.000256221;
   DATA[1233,13] := 1010.959;
   DATA[1233,14] := 1.0;
   DATA[1233,15] := 1.0;
   DATA[1233,16] := 1.0;
   DATA[1233,17] := 1.0;
   DATA[1233,18] := 1.0;
   DATA[1233,19] := 1.0;
   DATA[1233,20] := 148.808;
   DATA[1233,21] := 154.0374;
   DATA[1233,22] := 1.711082;
   DATA[1233,23] := 831.3253;
   DATA[1233,24] := 2.0;
   DATA[1233,25] := 2.0;
   DATA[1233,26] := 7.87798;
   DATA[1233,27] := 143.2966;
   DATA[1233,28] := 263.1056;
   DATA[1233,29] := 12.15073;
   DATA[1233,30] := 1.723404;
   DATA[1233,31] := 1.281798;
   DATA[1233,32] := 0.7352687;
   DATA[1233,33] := 0.3083624;
   DATA[1233,34] := 2.0;
   DATA[1233,35] := 250.016;
   DATA[1233,36] := 1.681991;
   DATA[1233,37] := 188.8138;
   DATA[1233,38] := 0.000128152;
   DATA[1233,39] := 1.0;
   DATA[1234,0] := 2.526022;
   DATA[1234,1] := 770.2961;
   DATA[1234,2] := 2.0;
   DATA[1234,3] := 1.0;
   DATA[1234,4] := 262.5288;
   DATA[1234,5] := 8.464048;
   DATA[1234,6] := 317.4058;
   DATA[1234,8] := 1.0;
   DATA[1234,9] := 1.0;
   DATA[1234,10] := 1.0;
   DATA[1234,11] := 2.010372;
   DATA[1234,12] := 0.000256221;
   DATA[1234,13] := 1010.879;
   DATA[1234,14] := 1.0;
   DATA[1234,15] := 1.0;
   DATA[1234,16] := 1.0;
   DATA[1234,17] := 1.0;
   DATA[1234,18] := 1.0;
   DATA[1234,19] := 1.0;
   DATA[1234,20] := 148.808;
   DATA[1234,21] := 154.0118;
   DATA[1234,22] := 1.711082;
   DATA[1234,23] := 830.8639;
   DATA[1234,24] := 2.0;
   DATA[1234,25] := 2.0;
   DATA[1234,26] := 7.87798;
   DATA[1234,27] := 143.2966;
   DATA[1234,28] := 263.1056;
   DATA[1234,29] := 12.15073;
   DATA[1234,30] := 1.723404;
   DATA[1234,31] := 1.281798;
   DATA[1234,32] := 0.7352687;
   DATA[1234,33] := 0.3083624;
   DATA[1234,34] := 2.0;
   DATA[1234,35] := 249.7757;
   DATA[1234,36] := 1.681991;
   DATA[1234,37] := 188.8138;
   DATA[1234,38] := 0.000128152;
   DATA[1234,39] := 1.0;
   DATA[1235,0] := 2.526022;
   DATA[1235,1] := 770.3746;
   DATA[1235,2] := 2.0;
   DATA[1235,3] := 1.0;
   DATA[1235,4] := 262.5288;
   DATA[1235,5] := 8.464048;
   DATA[1235,6] := 317.4058;
   DATA[1235,8] := 1.0;
   DATA[1235,9] := 1.0;
   DATA[1235,10] := 1.0;
   DATA[1235,11] := 2.010372;
   DATA[1235,12] := 0.000256221;
   DATA[1235,13] := 1010.638;
   DATA[1235,14] := 1.0;
   DATA[1235,15] := 1.0;
   DATA[1235,16] := 1.0;
   DATA[1235,17] := 1.0;
   DATA[1235,18] := 1.0;
   DATA[1235,19] := 1.0;
   DATA[1235,20] := 148.808;
   DATA[1235,21] := 154.0118;
   DATA[1235,22] := 1.711082;
   DATA[1235,23] := 830.6716;
   DATA[1235,24] := 2.0;
   DATA[1235,25] := 2.0;
   DATA[1235,26] := 7.87798;
   DATA[1235,27] := 143.2966;
   DATA[1235,28] := 263.1056;
   DATA[1235,29] := 12.11228;
   DATA[1235,30] := 1.723404;
   DATA[1235,31] := 1.281798;
   DATA[1235,32] := 0.7352687;
   DATA[1235,33] := 0.3083624;
   DATA[1235,34] := 2.0;
   DATA[1235,35] := 249.7757;
   DATA[1235,36] := 1.681991;
   DATA[1235,37] := 188.7016;
   DATA[1235,38] := 0.000128152;
   DATA[1235,39] := 1.0;
   DATA[1236,0] := 2.532748;
   DATA[1236,1] := 770.3746;
   DATA[1236,2] := 2.0;
   DATA[1236,3] := 1.0;
   DATA[1236,4] := 262.5288;
   DATA[1236,5] := 8.464048;
   DATA[1236,6] := 317.4058;
   DATA[1236,8] := 1.0;
   DATA[1236,9] := 1.0;
   DATA[1236,10] := 1.0;
   DATA[1236,11] := 2.010372;
   DATA[1236,12] := 0.000256221;
   DATA[1236,13] := 1010.758;
   DATA[1236,14] := 1.0;
   DATA[1236,15] := 1.0;
   DATA[1236,16] := 1.0;
   DATA[1236,17] := 1.0;
   DATA[1236,18] := 1.0;
   DATA[1236,19] := 1.0;
   DATA[1236,20] := 148.808;
   DATA[1236,21] := 154.0118;
   DATA[1236,22] := 1.711082;
   DATA[1236,23] := 830.2487;
   DATA[1236,24] := 2.0;
   DATA[1236,25] := 2.0;
   DATA[1236,26] := 7.87798;
   DATA[1236,27] := 143.2966;
   DATA[1236,28] := 263.1056;
   DATA[1236,29] := 12.11228;
   DATA[1236,30] := 1.723404;
   DATA[1236,31] := 1.281798;
   DATA[1236,32] := 0.7352687;
   DATA[1236,33] := 0.3083624;
   DATA[1236,34] := 2.0;
   DATA[1236,35] := 249.7757;
   DATA[1236,36] := 1.681991;
   DATA[1236,37] := 188.7016;
   DATA[1236,38] := 0.000128152;
   DATA[1236,39] := 1.0;
   DATA[1237,0] := 2.536912;
   DATA[1237,1] := 771.0027;
   DATA[1237,2] := 2.0;
   DATA[1237,3] := 1.0;
   DATA[1237,4] := 262.5288;
   DATA[1237,5] := 8.464048;
   DATA[1237,6] := 317.4058;
   DATA[1237,8] := 1.0;
   DATA[1237,9] := 1.0;
   DATA[1237,10] := 1.0;
   DATA[1237,11] := 2.010372;
   DATA[1237,12] := 0.000256221;
   DATA[1237,13] := 1011.039;
   DATA[1237,14] := 1.0;
   DATA[1237,15] := 1.0;
   DATA[1237,16] := 1.0;
   DATA[1237,17] := 1.0;
   DATA[1237,18] := 1.0;
   DATA[1237,19] := 1.0;
   DATA[1237,20] := 148.808;
   DATA[1237,21] := 154.0118;
   DATA[1237,22] := 1.710698;
   DATA[1237,23] := 830.2871;
   DATA[1237,24] := 2.0;
   DATA[1237,25] := 2.0;
   DATA[1237,26] := 7.87798;
   DATA[1237,27] := 143.2966;
   DATA[1237,28] := 263.1056;
   DATA[1237,29] := 12.11228;
   DATA[1237,30] := 1.721738;
   DATA[1237,31] := 1.278468;
   DATA[1237,32] := 0.7352687;
   DATA[1237,33] := 0.3083624;
   DATA[1237,34] := 2.0;
   DATA[1237,35] := 249.7757;
   DATA[1237,36] := 1.681991;
   DATA[1237,37] := 188.7016;
   DATA[1237,38] := 0.000128152;
   DATA[1237,39] := 1.0;
   DATA[1238,0] := 2.544919;
   DATA[1238,1] := 771.6307;
   DATA[1238,2] := 2.0;
   DATA[1238,3] := 1.0;
   DATA[1238,4] := 262.5288;
   DATA[1238,5] := 8.464048;
   DATA[1238,6] := 317.4058;
   DATA[1238,8] := 1.0;
   DATA[1238,9] := 1.0;
   DATA[1238,10] := 1.0;
   DATA[1238,11] := 2.010372;
   DATA[1238,12] := 0.000256221;
   DATA[1238,13] := 1010.718;
   DATA[1238,14] := 1.0;
   DATA[1238,15] := 1.0;
   DATA[1238,16] := 1.0;
   DATA[1238,17] := 1.0;
   DATA[1238,18] := 1.0;
   DATA[1238,19] := 1.0;
   DATA[1238,20] := 148.808;
   DATA[1238,21] := 154.0118;
   DATA[1238,22] := 1.710698;
   DATA[1238,23] := 829.9026;
   DATA[1238,24] := 2.0;
   DATA[1238,25] := 2.0;
   DATA[1238,26] := 7.87798;
   DATA[1238,27] := 143.2966;
   DATA[1238,28] := 263.1056;
   DATA[1238,29] := 12.11228;
   DATA[1238,30] := 1.721738;
   DATA[1238,31] := 1.275138;
   DATA[1238,32] := 0.7352687;
   DATA[1238,33] := 0.3083624;
   DATA[1238,34] := 2.0;
   DATA[1238,35] := 249.984;
   DATA[1238,36] := 1.681991;
   DATA[1238,37] := 188.7016;
   DATA[1238,38] := 0.000128152;
   DATA[1238,39] := 1.0;
   DATA[1239,0] := 2.547161;
   DATA[1239,1] := 771.9448;
   DATA[1239,2] := 2.0;
   DATA[1239,3] := 1.0;
   DATA[1239,4] := 262.5288;
   DATA[1239,5] := 8.467573;
   DATA[1239,6] := 317.4058;
   DATA[1239,8] := 1.0;
   DATA[1239,9] := 1.0;
   DATA[1239,10] := 1.0;
   DATA[1239,11] := 2.010372;
   DATA[1239,12] := 0.000256221;
   DATA[1239,13] := 1011.039;
   DATA[1239,14] := 1.0;
   DATA[1239,15] := 1.0;
   DATA[1239,16] := 1.0;
   DATA[1239,17] := 1.0;
   DATA[1239,18] := 1.0;
   DATA[1239,19] := 1.0;
   DATA[1239,20] := 148.808;
   DATA[1239,21] := 154.14;
   DATA[1239,22] := 1.710698;
   DATA[1239,23] := 829.2874;
   DATA[1239,24] := 2.0;
   DATA[1239,25] := 2.0;
   DATA[1239,26] := 7.87798;
   DATA[1239,27] := 143.2966;
   DATA[1239,28] := 263.1056;
   DATA[1239,29] := 12.11228;
   DATA[1239,30] := 1.721738;
   DATA[1239,31] := 1.277059;
   DATA[1239,32] := 0.7352687;
   DATA[1239,33] := 0.3083624;
   DATA[1239,34] := 2.0;
   DATA[1239,35] := 249.984;
   DATA[1239,36] := 1.681991;
   DATA[1239,37] := 188.7337;
   DATA[1239,38] := 0.000128152;
   DATA[1239,39] := 1.0;
   DATA[1240,0] := 2.548442;
   DATA[1240,1] := 772.769;
   DATA[1240,2] := 2.0;
   DATA[1240,3] := 1.0;
   DATA[1240,4] := 262.5288;
   DATA[1240,5] := 8.467573;
   DATA[1240,6] := 317.4058;
   DATA[1240,8] := 1.0;
   DATA[1240,9] := 1.0;
   DATA[1240,10] := 1.0;
   DATA[1240,11] := 2.010372;
   DATA[1240,12] := 0.000256221;
   DATA[1240,13] := 1011.359;
   DATA[1240,14] := 1.0;
   DATA[1240,15] := 1.0;
   DATA[1240,16] := 1.0;
   DATA[1240,17] := 1.0;
   DATA[1240,18] := 1.0;
   DATA[1240,19] := 1.0;
   DATA[1240,20] := 148.808;
   DATA[1240,21] := 154.14;
   DATA[1240,22] := 1.710698;
   DATA[1240,23] := 829.1335;
   DATA[1240,24] := 2.0;
   DATA[1240,25] := 2.0;
   DATA[1240,26] := 7.87798;
   DATA[1240,27] := 143.2966;
   DATA[1240,28] := 263.1056;
   DATA[1240,29] := 12.11228;
   DATA[1240,30] := 1.721738;
   DATA[1240,31] := 1.270911;
   DATA[1240,32] := 0.7352687;
   DATA[1240,33] := 0.3083624;
   DATA[1240,34] := 2.0;
   DATA[1240,35] := 249.984;
   DATA[1240,36] := 1.681991;
   DATA[1240,37] := 188.8138;
   DATA[1240,38] := 0.000128152;
   DATA[1240,39] := 1.0;
   DATA[1241,0] := 2.550043;
   DATA[1241,1] := 773.3971;
   DATA[1241,2] := 2.0;
   DATA[1241,3] := 1.0;
   DATA[1241,4] := 262.5288;
   DATA[1241,5] := 8.467573;
   DATA[1241,6] := 317.4058;
   DATA[1241,8] := 1.0;
   DATA[1241,9] := 1.0;
   DATA[1241,10] := 1.0;
   DATA[1241,11] := 2.010372;
   DATA[1241,12] := 0.000256221;
   DATA[1241,13] := 1011.119;
   DATA[1241,14] := 1.0;
   DATA[1241,15] := 1.0;
   DATA[1241,16] := 1.0;
   DATA[1241,17] := 1.0;
   DATA[1241,18] := 1.0;
   DATA[1241,19] := 1.0;
   DATA[1241,20] := 148.808;
   DATA[1241,21] := 154.14;
   DATA[1241,22] := 1.713004;
   DATA[1241,23] := 828.5183;
   DATA[1241,24] := 2.0;
   DATA[1241,25] := 2.0;
   DATA[1241,26] := 7.87798;
   DATA[1241,27] := 143.2966;
   DATA[1241,28] := 263.1056;
   DATA[1241,29] := 12.11228;
   DATA[1241,30] := 1.721482;
   DATA[1241,31] := 1.274625;
   DATA[1241,32] := 0.7352687;
   DATA[1241,33] := 0.3104122;
   DATA[1241,34] := 2.0;
   DATA[1241,35] := 249.984;
   DATA[1241,36] := 1.681991;
   DATA[1241,37] := 188.8939;
   DATA[1241,38] := 0.000128152;
   DATA[1241,39] := 1.0;
   DATA[1242,0] := 2.541716;
   DATA[1242,1] := 773.9467;
   DATA[1242,2] := 2.0;
   DATA[1242,3] := 1.0;
   DATA[1242,4] := 262.5288;
   DATA[1242,5] := 8.467573;
   DATA[1242,6] := 317.4058;
   DATA[1242,8] := 1.0;
   DATA[1242,9] := 1.0;
   DATA[1242,10] := 1.0;
   DATA[1242,11] := 2.010372;
   DATA[1242,12] := 0.000256221;
   DATA[1242,13] := 1011.119;
   DATA[1242,14] := 1.0;
   DATA[1242,15] := 1.0;
   DATA[1242,16] := 1.0;
   DATA[1242,17] := 1.0;
   DATA[1242,18] := 1.0;
   DATA[1242,19] := 1.0;
   DATA[1242,20] := 148.808;
   DATA[1242,21] := 154.14;
   DATA[1242,22] := 1.714029;
   DATA[1242,23] := 828.5568;
   DATA[1242,24] := 2.0;
   DATA[1242,25] := 2.0;
   DATA[1242,26] := 7.87798;
   DATA[1242,27] := 143.2966;
   DATA[1242,28] := 263.1056;
   DATA[1242,29] := 12.11228;
   DATA[1242,30] := 1.721482;
   DATA[1242,31] := 1.276803;
   DATA[1242,32] := 0.7352687;
   DATA[1242,33] := 0.3106043;
   DATA[1242,34] := 2.0;
   DATA[1242,35] := 249.984;
   DATA[1242,36] := 1.681991;
   DATA[1242,37] := 188.8939;
   DATA[1242,38] := 0.000128152;
   DATA[1242,39] := 1.0;
   DATA[1243,0] := 2.538513;
   DATA[1243,1] := 774.1821;
   DATA[1243,2] := 2.0;
   DATA[1243,3] := 1.0;
   DATA[1243,4] := 262.5288;
   DATA[1243,5] := 8.467573;
   DATA[1243,6] := 317.4058;
   DATA[1243,8] := 1.0;
   DATA[1243,9] := 1.0;
   DATA[1243,10] := 1.0;
   DATA[1243,11] := 2.010372;
   DATA[1243,12] := 0.000256221;
   DATA[1243,13] := 1011.079;
   DATA[1243,14] := 1.0;
   DATA[1243,15] := 1.0;
   DATA[1243,16] := 1.0;
   DATA[1243,17] := 1.0;
   DATA[1243,18] := 1.0;
   DATA[1243,19] := 1.0;
   DATA[1243,20] := 148.808;
   DATA[1243,21] := 154.14;
   DATA[1243,22] := 1.714798;
   DATA[1243,23] := 828.0569;
   DATA[1243,24] := 2.0;
   DATA[1243,25] := 2.0;
   DATA[1243,26] := 7.878621;
   DATA[1243,27] := 143.2966;
   DATA[1243,28] := 263.1056;
   DATA[1243,29] := 12.11228;
   DATA[1243,30] := 1.721482;
   DATA[1243,31] := 1.277956;
   DATA[1243,32] := 0.7352687;
   DATA[1243,33] := 0.3093233;
   DATA[1243,34] := 2.0;
   DATA[1243,35] := 249.984;
   DATA[1243,36] := 1.681991;
   DATA[1243,37] := 188.8939;
   DATA[1243,38] := 0.000128152;
   DATA[1243,39] := 1.0;
   DATA[1244,0] := 2.535951;
   DATA[1244,1] := 774.6924;
   DATA[1244,2] := 2.0;
   DATA[1244,3] := 1.0;
   DATA[1244,4] := 262.5288;
   DATA[1244,5] := 8.467573;
   DATA[1244,6] := 317.4058;
   DATA[1244,8] := 1.0;
   DATA[1244,9] := 1.0;
   DATA[1244,10] := 1.0;
   DATA[1244,11] := 2.010372;
   DATA[1244,12] := 0.000256221;
   DATA[1244,13] := 1011.359;
   DATA[1244,14] := 1.0;
   DATA[1244,15] := 1.0;
   DATA[1244,16] := 1.0;
   DATA[1244,17] := 1.0;
   DATA[1244,18] := 1.0;
   DATA[1244,19] := 1.0;
   DATA[1244,20] := 148.808;
   DATA[1244,21] := 154.14;
   DATA[1244,22] := 1.714798;
   DATA[1244,23] := 827.8646;
   DATA[1244,24] := 2.0;
   DATA[1244,25] := 2.0;
   DATA[1244,26] := 7.879262;
   DATA[1244,27] := 143.2966;
   DATA[1244,28] := 263.1056;
   DATA[1244,29] := 12.11228;
   DATA[1244,30] := 1.721482;
   DATA[1244,31] := 1.281927;
   DATA[1244,32] := 0.7352687;
   DATA[1244,33] := 0.3093233;
   DATA[1244,34] := 2.0;
   DATA[1244,35] := 249.984;
   DATA[1244,36] := 1.681991;
   DATA[1244,37] := 188.8939;
   DATA[1244,38] := 0.000128152;
   DATA[1244,39] := 1.0;
   DATA[1245,0] := 2.535951;
   DATA[1245,1] := 775.2813;
   DATA[1245,2] := 2.0;
   DATA[1245,3] := 1.0;
   DATA[1245,4] := 262.5288;
   DATA[1245,5] := 8.467573;
   DATA[1245,6] := 317.4058;
   DATA[1245,8] := 1.0;
   DATA[1245,9] := 1.0;
   DATA[1245,10] := 1.0;
   DATA[1245,11] := 2.010372;
   DATA[1245,12] := 0.000256221;
   DATA[1245,13] := 1011.279;
   DATA[1245,14] := 1.0;
   DATA[1245,15] := 1.0;
   DATA[1245,16] := 1.0;
   DATA[1245,17] := 1.0;
   DATA[1245,18] := 1.0;
   DATA[1245,19] := 1.0;
   DATA[1245,20] := 148.808;
   DATA[1245,21] := 154.14;
   DATA[1245,22] := 1.711595;
   DATA[1245,23] := 827.2879;
   DATA[1245,24] := 2.0;
   DATA[1245,25] := 2.0;
   DATA[1245,26] := 7.879262;
   DATA[1245,27] := 143.2966;
   DATA[1245,28] := 263.1056;
   DATA[1245,29] := 12.11228;
   DATA[1245,30] := 1.72443;
   DATA[1245,31] := 1.281927;
   DATA[1245,32] := 0.7352687;
   DATA[1245,33] := 0.3106684;
   DATA[1245,34] := 2.0;
   DATA[1245,35] := 249.984;
   DATA[1245,36] := 1.617916;
   DATA[1245,37] := 188.7176;
   DATA[1245,38] := 0.000128152;
   DATA[1245,39] := 1.0;
   DATA[1246,0] := 2.535951;
   DATA[1246,1] := 775.87;
   DATA[1246,2] := 2.0;
   DATA[1246,3] := 1.0;
   DATA[1246,4] := 262.5288;
   DATA[1246,5] := 8.467573;
   DATA[1246,6] := 317.4058;
   DATA[1246,8] := 1.0;
   DATA[1246,9] := 1.0;
   DATA[1246,10] := 1.0;
   DATA[1246,11] := 2.010372;
   DATA[1246,12] := 0.000256221;
   DATA[1246,13] := 1010.959;
   DATA[1246,14] := 1.0;
   DATA[1246,15] := 1.0;
   DATA[1246,16] := 1.0;
   DATA[1246,17] := 1.0;
   DATA[1246,18] := 1.0;
   DATA[1246,19] := 1.0;
   DATA[1246,20] := 148.808;
   DATA[1246,21] := 154.14;
   DATA[1246,22] := 1.711338;
   DATA[1246,23] := 826.9418;
   DATA[1246,24] := 2.0;
   DATA[1246,25] := 2.0;
   DATA[1246,26] := 7.879262;
   DATA[1246,27] := 143.2966;
   DATA[1246,28] := 263.1056;
   DATA[1246,29] := 12.11228;
   DATA[1246,30] := 1.72443;
   DATA[1246,31] := 1.289228;
   DATA[1246,32] := 0.7352687;
   DATA[1246,33] := 0.3106684;
   DATA[1246,34] := 2.0;
   DATA[1246,35] := 249.984;
   DATA[1246,36] := 1.617916;
   DATA[1246,37] := 188.7176;
   DATA[1246,38] := 0.000128152;
   DATA[1246,39] := 1.0;
   DATA[1247,0] := 2.535951;
   DATA[1247,1] := 776.6551;
   DATA[1247,2] := 2.0;
   DATA[1247,3] := 1.0;
   DATA[1247,4] := 262.5288;
   DATA[1247,5] := 8.467573;
   DATA[1247,6] := 317.4058;
   DATA[1247,8] := 1.0;
   DATA[1247,9] := 1.0;
   DATA[1247,10] := 1.0;
   DATA[1247,11] := 2.010372;
   DATA[1247,12] := 0.000256221;
   DATA[1247,13] := 1011.039;
   DATA[1247,14] := 1.0;
   DATA[1247,15] := 1.0;
   DATA[1247,16] := 1.0;
   DATA[1247,17] := 1.0;
   DATA[1247,18] := 1.0;
   DATA[1247,19] := 1.0;
   DATA[1247,20] := 148.808;
   DATA[1247,21] := 154.14;
   DATA[1247,22] := 1.711338;
   DATA[1247,23] := 826.5573;
   DATA[1247,24] := 2.0;
   DATA[1247,25] := 2.0;
   DATA[1247,26] := 7.879262;
   DATA[1247,27] := 143.2966;
   DATA[1247,28] := 263.1056;
   DATA[1247,29] := 12.11228;
   DATA[1247,30] := 1.722251;
   DATA[1247,31] := 1.291533;
   DATA[1247,32] := 0.7352687;
   DATA[1247,33] := 0.3106684;
   DATA[1247,34] := 2.0;
   DATA[1247,35] := 249.8398;
   DATA[1247,36] := 1.617916;
   DATA[1247,37] := 188.7176;
   DATA[1247,38] := 0.000128152;
   DATA[1247,39] := 1.0;
   DATA[1248,0] := 2.535951;
   DATA[1248,1] := 777.3616;
   DATA[1248,2] := 2.0;
   DATA[1248,3] := 1.0;
   DATA[1248,4] := 262.5288;
   DATA[1248,5] := 8.469175;
   DATA[1248,6] := 317.4058;
   DATA[1248,8] := 1.0;
   DATA[1248,9] := 1.0;
   DATA[1248,10] := 1.0;
   DATA[1248,11] := 2.010372;
   DATA[1248,12] := 0.000256221;
   DATA[1248,13] := 1010.959;
   DATA[1248,14] := 1.0;
   DATA[1248,15] := 1.0;
   DATA[1248,16] := 1.0;
   DATA[1248,17] := 1.0;
   DATA[1248,18] := 1.0;
   DATA[1248,19] := 1.0;
   DATA[1248,20] := 148.808;
   DATA[1248,21] := 154.14;
   DATA[1248,22] := 1.711338;
   DATA[1248,23] := 826.4035;
   DATA[1248,24] := 2.0;
   DATA[1248,25] := 2.0;
   DATA[1248,26] := 7.879262;
   DATA[1248,27] := 143.2966;
   DATA[1248,28] := 263.1056;
   DATA[1248,29] := 12.11228;
   DATA[1248,30] := 1.721738;
   DATA[1248,31] := 1.291533;
   DATA[1248,32] := 0.7352687;
   DATA[1248,33] := 0.309067;
   DATA[1248,34] := 2.0;
   DATA[1248,35] := 249.7437;
   DATA[1248,36] := 1.617916;
   DATA[1248,37] := 188.6055;
   DATA[1248,38] := 0.000128152;
   DATA[1248,39] := 1.0;
   DATA[1249,0] := 2.538833;
   DATA[1249,1] := 777.6364;
   DATA[1249,2] := 2.0;
   DATA[1249,3] := 1.0;
   DATA[1249,4] := 262.5288;
   DATA[1249,5] := 8.470457;
   DATA[1249,6] := 317.4058;
   DATA[1249,8] := 1.0;
   DATA[1249,9] := 1.0;
   DATA[1249,10] := 1.0;
   DATA[1249,11] := 2.010372;
   DATA[1249,13] := 1011.039;
   DATA[1249,14] := 1.0;
   DATA[1249,15] := 1.0;
   DATA[1249,16] := 1.0;
   DATA[1249,17] := 1.0;
   DATA[1249,18] := 1.0;
   DATA[1249,19] := 1.0;
   DATA[1249,20] := 148.808;
   DATA[1249,21] := 154.14;
   DATA[1249,22] := 1.710954;
   DATA[1249,23] := 826.4035;
   DATA[1249,24] := 2.0;
   DATA[1249,25] := 2.0;
   DATA[1249,26] := 7.879262;
   DATA[1249,27] := 143.1684;
   DATA[1249,28] := 263.1056;
   DATA[1249,29] := 11.95847;
   DATA[1249,30] := 1.721738;
   DATA[1249,31] := 1.290124;
   DATA[1249,32] := 0.7352687;
   DATA[1249,33] := 0.3088108;
   DATA[1249,34] := 2.0;
   DATA[1249,35] := 249.7437;
   DATA[1249,36] := 1.617916;
   DATA[1249,37] := 188.6055;
   DATA[1249,38] := 0.000128152;
   DATA[1249,39] := 1.0;
   DATA[1250,0] := 2.543958;
   DATA[1250,1] := 778.3037;
   DATA[1250,2] := 2.0;
   DATA[1250,3] := 1.0;
   DATA[1250,4] := 262.5288;
   DATA[1250,5] := 8.470457;
   DATA[1250,6] := 317.4058;
   DATA[1250,8] := 1.0;
   DATA[1250,9] := 1.0;
   DATA[1250,10] := 1.0;
   DATA[1250,11] := 2.010372;
   DATA[1250,13] := 1010.718;
   DATA[1250,14] := 1.0;
   DATA[1250,15] := 1.0;
   DATA[1250,16] := 1.0;
   DATA[1250,17] := 1.0;
   DATA[1250,18] := 1.0;
   DATA[1250,19] := 1.0;
   DATA[1250,20] := 148.808;
   DATA[1250,21] := 154.14;
   DATA[1250,22] := 1.708391;
   DATA[1250,23] := 825.9421;
   DATA[1250,24] := 2.0;
   DATA[1250,25] := 2.0;
   DATA[1250,26] := 7.879262;
   DATA[1250,27] := 143.1684;
   DATA[1250,28] := 263.1056;
   DATA[1250,29] := 11.95847;
   DATA[1250,30] := 1.721738;
   DATA[1250,31] := 1.273345;
   DATA[1250,32] := 0.7352687;
   DATA[1250,33] := 0.3086186;
   DATA[1250,34] := 2.0;
   DATA[1250,35] := 249.7437;
   DATA[1250,36] := 1.617916;
   DATA[1250,37] := 188.6055;
   DATA[1250,38] := 0.000128152;
   DATA[1250,39] := 1.0;
   DATA[1251,0] := 2.54588;
   DATA[1251,1] := 779.0495;
   DATA[1251,2] := 2.0;
   DATA[1251,3] := 1.0;
   DATA[1251,4] := 262.5288;
   DATA[1251,5] := 8.467253;
   DATA[1251,6] := 317.4058;
   DATA[1251,8] := 1.0;
   DATA[1251,9] := 1.0;
   DATA[1251,10] := 1.0;
   DATA[1251,11] := 2.010372;
   DATA[1251,13] := 1010.919;
   DATA[1251,14] := 1.0;
   DATA[1251,15] := 1.0;
   DATA[1251,16] := 1.0;
   DATA[1251,17] := 1.0;
   DATA[1251,18] := 1.0;
   DATA[1251,19] := 1.0;
   DATA[1251,20] := 148.808;
   DATA[1251,21] := 154.14;
   DATA[1251,22] := 1.708263;
   DATA[1251,23] := 825.4422;
   DATA[1251,24] := 2.0;
   DATA[1251,25] := 2.0;
   DATA[1251,26] := 7.879262;
   DATA[1251,27] := 143.1684;
   DATA[1251,28] := 263.1056;
   DATA[1251,29] := 11.95847;
   DATA[1251,30] := 1.721738;
   DATA[1251,31] := 1.27834;
   DATA[1251,32] := 0.7352687;
   DATA[1251,33] := 0.3086186;
   DATA[1251,34] := 2.0;
   DATA[1251,35] := 250.0;
   DATA[1251,36] := 1.617916;
   DATA[1251,37] := 188.7016;
   DATA[1251,38] := 0.000128152;
   DATA[1251,39] := 1.0;
   DATA[1252,0] := 2.548442;
   DATA[1252,1] := 779.442;
   DATA[1252,2] := 2.0;
   DATA[1252,3] := 1.0;
   DATA[1252,4] := 262.5288;
   DATA[1252,5] := 8.46533;
   DATA[1252,6] := 317.5596;
   DATA[1252,8] := 1.0;
   DATA[1252,9] := 1.0;
   DATA[1252,10] := 1.0;
   DATA[1252,11] := 2.010372;
   DATA[1252,13] := 1011.079;
   DATA[1252,14] := 1.0;
   DATA[1252,15] := 1.0;
   DATA[1252,16] := 1.0;
   DATA[1252,17] := 1.0;
   DATA[1252,18] := 1.0;
   DATA[1252,19] := 1.0;
   DATA[1252,20] := 148.808;
   DATA[1252,21] := 154.14;
   DATA[1252,22] := 1.709672;
   DATA[1252,23] := 825.173;
   DATA[1252,24] := 2.0;
   DATA[1252,25] := 2.0;
   DATA[1252,26] := 7.879262;
   DATA[1252,27] := 143.1684;
   DATA[1252,28] := 262.8172;
   DATA[1252,29] := 11.95847;
   DATA[1252,30] := 1.721738;
   DATA[1252,31] := 1.281158;
   DATA[1252,32] := 0.7360369;
   DATA[1252,33] := 0.3084905;
   DATA[1252,34] := 2.0;
   DATA[1252,35] := 250.0;
   DATA[1252,36] := 1.617916;
   DATA[1252,37] := 188.7817;
   DATA[1252,38] := 0.000128152;
   DATA[1252,39] := 1.0;
   DATA[1253,0] := 2.548442;
   DATA[1253,1] := 779.6383;
   DATA[1253,2] := 2.0;
   DATA[1253,3] := 1.0;
   DATA[1253,4] := 262.5288;
   DATA[1253,5] := 8.464369;
   DATA[1253,6] := 317.5596;
   DATA[1253,8] := 1.0;
   DATA[1253,9] := 1.0;
   DATA[1253,10] := 1.0;
   DATA[1253,11] := 2.010372;
   DATA[1253,13] := 1011.079;
   DATA[1253,14] := 1.0;
   DATA[1253,15] := 1.0;
   DATA[1253,16] := 1.0;
   DATA[1253,17] := 1.0;
   DATA[1253,18] := 1.0;
   DATA[1253,19] := 1.0;
   DATA[1253,20] := 148.808;
   DATA[1253,21] := 154.14;
   DATA[1253,22] := 1.711338;
   DATA[1253,23] := 824.8654;
   DATA[1253,24] := 2.0;
   DATA[1253,25] := 2.0;
   DATA[1253,26] := 7.879262;
   DATA[1253,27] := 143.1684;
   DATA[1253,28] := 262.8172;
   DATA[1253,29] := 11.95847;
   DATA[1253,30] := 1.721738;
   DATA[1253,31] := 1.281158;
   DATA[1253,32] := 0.7360369;
   DATA[1253,33] := 0.3082983;
   DATA[1253,34] := 2.0;
   DATA[1253,35] := 250.0;
   DATA[1253,36] := 1.617916;
   DATA[1253,37] := 188.8939;
   DATA[1253,38] := 0.000128152;
   DATA[1253,39] := 1.0;
   DATA[1254,0] := 2.548442;
   DATA[1254,1] := 779.913;
   DATA[1254,2] := 2.0;
   DATA[1254,3] := 1.0;
   DATA[1254,4] := 262.5288;
   DATA[1254,5] := 8.464369;
   DATA[1254,6] := 317.5596;
   DATA[1254,8] := 1.0;
   DATA[1254,9] := 1.0;
   DATA[1254,10] := 1.0;
   DATA[1254,11] := 2.010372;
   DATA[1254,12] := 0.000384332;
   DATA[1254,13] := 1010.879;
   DATA[1254,14] := 1.0;
   DATA[1254,15] := 1.0;
   DATA[1254,16] := 1.0;
   DATA[1254,17] := 1.0;
   DATA[1254,18] := 1.0;
   DATA[1254,19] := 1.0;
   DATA[1254,20] := 148.808;
   DATA[1254,21] := 154.14;
   DATA[1254,22] := 1.711338;
   DATA[1254,23] := 824.4809;
   DATA[1254,24] := 2.0;
   DATA[1254,25] := 2.0;
   DATA[1254,26] := 7.877019;
   DATA[1254,27] := 143.1684;
   DATA[1254,28] := 262.8172;
   DATA[1254,29] := 11.95847;
   DATA[1254,30] := 1.72443;
   DATA[1254,31] := 1.282823;
   DATA[1254,32] := 0.7360369;
   DATA[1254,33] := 0.3082983;
   DATA[1254,34] := 2.0;
   DATA[1254,35] := 250.1122;
   DATA[1254,36] := 1.617916;
   DATA[1254,37] := 188.8939;
   DATA[1254,38] := 0.000128152;
   DATA[1254,39] := 1.0;
   DATA[1255,0] := 2.548442;
   DATA[1255,1] := 780.3841;
   DATA[1255,2] := 2.0;
   DATA[1255,3] := 1.0;
   DATA[1255,4] := 262.5288;
   DATA[1255,5] := 8.464369;
   DATA[1255,6] := 317.5596;
   DATA[1255,8] := 1.0;
   DATA[1255,9] := 1.0;
   DATA[1255,10] := 1.0;
   DATA[1255,11] := 2.010372;
   DATA[1255,12] := 0.000384332;
   DATA[1255,13] := 1010.758;
   DATA[1255,14] := 1.0;
   DATA[1255,15] := 1.0;
   DATA[1255,16] := 1.0;
   DATA[1255,17] := 1.0;
   DATA[1255,18] := 1.0;
   DATA[1255,19] := 1.0;
   DATA[1255,20] := 148.808;
   DATA[1255,21] := 154.14;
   DATA[1255,22] := 1.711338;
   DATA[1255,23] := 824.0964;
   DATA[1255,24] := 2.0;
   DATA[1255,25] := 2.0;
   DATA[1255,26] := 7.877019;
   DATA[1255,27] := 143.1684;
   DATA[1255,28] := 262.8172;
   DATA[1255,29] := 12.03538;
   DATA[1255,30] := 1.72443;
   DATA[1255,31] := 1.282823;
   DATA[1255,32] := 0.7360369;
   DATA[1255,33] := 0.3082983;
   DATA[1255,34] := 2.0;
   DATA[1255,35] := 250.1762;
   DATA[1255,36] := 1.617916;
   DATA[1255,37] := 188.8939;
   DATA[1255,38] := 0.000128152;
   DATA[1255,39] := 1.0;
   DATA[1256,0] := 2.543638;
   DATA[1256,1] := 780.7766;
   DATA[1256,2] := 2.0;
   DATA[1256,3] := 1.0;
   DATA[1256,4] := 262.5288;
   DATA[1256,5] := 8.464369;
   DATA[1256,6] := 317.5596;
   DATA[1256,8] := 1.0;
   DATA[1256,9] := 1.0;
   DATA[1256,10] := 1.0;
   DATA[1256,11] := 2.010372;
   DATA[1256,12] := 0.000384332;
   DATA[1256,13] := 1010.718;
   DATA[1256,14] := 1.0;
   DATA[1256,15] := 1.0;
   DATA[1256,16] := 1.0;
   DATA[1256,17] := 1.0;
   DATA[1256,18] := 1.0;
   DATA[1256,19] := 1.0;
   DATA[1256,20] := 148.808;
   DATA[1256,21] := 154.14;
   DATA[1256,22] := 1.712363;
   DATA[1256,23] := 823.7119;
   DATA[1256,24] := 2.0;
   DATA[1256,25] := 2.0;
   DATA[1256,26] := 7.877019;
   DATA[1256,27] := 143.1684;
   DATA[1256,28] := 263.0095;
   DATA[1256,29] := 12.03538;
   DATA[1256,30] := 1.72443;
   DATA[1256,31] := 1.275138;
   DATA[1256,32] := 0.7352687;
   DATA[1256,33] := 0.3082983;
   DATA[1256,34] := 2.0;
   DATA[1256,35] := 250.1762;
   DATA[1256,36] := 1.617916;
   DATA[1256,37] := 189.1022;
   DATA[1256,38] := 0.000128152;
   DATA[1256,39] := 1.0;
   DATA[1257,0] := 2.541716;
   DATA[1257,1] := 781.4047;
   DATA[1257,2] := 2.0;
   DATA[1257,3] := 1.0;
   DATA[1257,4] := 262.5288;
   DATA[1257,5] := 8.464369;
   DATA[1257,6] := 317.5596;
   DATA[1257,8] := 1.0;
   DATA[1257,9] := 1.0;
   DATA[1257,10] := 1.0;
   DATA[1257,11] := 2.010372;
   DATA[1257,12] := 0.000384332;
   DATA[1257,13] := 1010.638;
   DATA[1257,14] := 1.0;
   DATA[1257,15] := 1.0;
   DATA[1257,16] := 1.0;
   DATA[1257,17] := 1.0;
   DATA[1257,18] := 1.0;
   DATA[1257,19] := 1.0;
   DATA[1257,20] := 148.808;
   DATA[1257,21] := 154.14;
   DATA[1257,22] := 1.71467;
   DATA[1257,23] := 823.3273;
   DATA[1257,24] := 2.0;
   DATA[1257,25] := 2.0;
   DATA[1257,26] := 7.87798;
   DATA[1257,27] := 143.1684;
   DATA[1257,28] := 263.0095;
   DATA[1257,29] := 12.03538;
   DATA[1257,30] := 1.725455;
   DATA[1257,31] := 1.261432;
   DATA[1257,32] := 0.7352687;
   DATA[1257,33] := 0.3082983;
   DATA[1257,34] := 2.0;
   DATA[1257,35] := 250.1762;
   DATA[1257,36] := 1.69801;
   DATA[1257,37] := 189.1022;
   DATA[1257,38] := 0.000128152;
   DATA[1257,39] := 1.0;
   DATA[1258,0] := 2.536912;
   DATA[1258,1] := 781.5616;
   DATA[1258,2] := 2.0;
   DATA[1258,3] := 1.0;
   DATA[1258,4] := 262.5288;
   DATA[1258,5] := 8.464369;
   DATA[1258,6] := 317.5596;
   DATA[1258,8] := 1.0;
   DATA[1258,9] := 1.0;
   DATA[1258,10] := 1.0;
   DATA[1258,11] := 2.010372;
   DATA[1258,12] := 0.000384332;
   DATA[1258,13] := 1010.678;
   DATA[1258,14] := 1.0;
   DATA[1258,15] := 1.0;
   DATA[1258,16] := 1.0;
   DATA[1258,17] := 1.0;
   DATA[1258,18] := 1.0;
   DATA[1258,19] := 1.0;
   DATA[1258,20] := 148.808;
   DATA[1258,21] := 154.14;
   DATA[1258,22] := 1.715183;
   DATA[1258,23] := 822.4814;
   DATA[1258,24] := 2.0;
   DATA[1258,25] := 2.0;
   DATA[1258,26] := 7.87798;
   DATA[1258,27] := 143.1684;
   DATA[1258,28] := 263.0095;
   DATA[1258,29] := 12.15073;
   DATA[1258,30] := 1.726096;
   DATA[1258,31] := 1.269758;
   DATA[1258,32] := 0.7352687;
   DATA[1258,33] := 0.3082983;
   DATA[1258,34] := 2.0;
   DATA[1258,35] := 250.1762;
   DATA[1258,36] := 1.69801;
   DATA[1258,37] := 189.1022;
   DATA[1258,38] := 0.000128152;
   DATA[1258,39] := 1.0;
   DATA[1259,0] := 2.532108;
   DATA[1259,1] := 782.2289;
   DATA[1259,2] := 2.0;
   DATA[1259,3] := 1.0;
   DATA[1259,4] := 262.5288;
   DATA[1259,5] := 8.464369;
   DATA[1259,6] := 317.4827;
   DATA[1259,8] := 1.0;
   DATA[1259,9] := 1.0;
   DATA[1259,10] := 1.0;
   DATA[1259,11] := 2.010372;
   DATA[1259,12] := 0.000384332;
   DATA[1259,13] := 1010.959;
   DATA[1259,14] := 1.0;
   DATA[1259,15] := 1.0;
   DATA[1259,16] := 1.0;
   DATA[1259,17] := 1.0;
   DATA[1259,18] := 1.0;
   DATA[1259,19] := 1.0;
   DATA[1259,20] := 148.808;
   DATA[1259,21] := 154.14;
   DATA[1259,22] := 1.715183;
   DATA[1259,23] := 822.4814;
   DATA[1259,24] := 2.0;
   DATA[1259,25] := 2.0;
   DATA[1259,26] := 7.87798;
   DATA[1259,27] := 142.9377;
   DATA[1259,28] := 263.0095;
   DATA[1259,29] := 12.15073;
   DATA[1259,30] := 1.726096;
   DATA[1259,31] := 1.271551;
   DATA[1259,32] := 0.7352687;
   DATA[1259,33] := 0.3082983;
   DATA[1259,34] := 2.0;
   DATA[1259,35] := 250.1762;
   DATA[1259,36] := 1.69801;
   DATA[1259,37] := 189.1022;
   DATA[1259,38] := 0.000128152;
   DATA[1259,39] := 1.0;
   DATA[1260,0] := 2.531467;
   DATA[1260,1] := 782.7393;
   DATA[1260,2] := 2.0;
   DATA[1260,3] := 1.0;
   DATA[1260,4] := 262.5288;
   DATA[1260,5] := 8.464369;
   DATA[1260,6] := 317.4827;
   DATA[1260,8] := 1.0;
   DATA[1260,9] := 1.0;
   DATA[1260,10] := 1.0;
   DATA[1260,11] := 2.010372;
   DATA[1260,13] := 1011.239;
   DATA[1260,14] := 1.0;
   DATA[1260,15] := 1.0;
   DATA[1260,16] := 1.0;
   DATA[1260,17] := 1.0;
   DATA[1260,18] := 1.0;
   DATA[1260,19] := 1.0;
   DATA[1260,20] := 148.808;
   DATA[1260,21] := 154.14;
   DATA[1260,22] := 1.715952;
   DATA[1260,23] := 821.9816;
   DATA[1260,24] := 2.0;
   DATA[1260,25] := 2.0;
   DATA[1260,26] := 7.87798;
   DATA[1260,27] := 142.9377;
   DATA[1260,28] := 263.0095;
   DATA[1260,29] := 12.15073;
   DATA[1260,30] := 1.726096;
   DATA[1260,31] := 1.272192;
   DATA[1260,32] := 0.7352687;
   DATA[1260,33] := 0.3082983;
   DATA[1260,34] := 2.0;
   DATA[1260,35] := 250.1762;
   DATA[1260,36] := 1.69801;
   DATA[1260,37] := 189.1022;
   DATA[1260,38] := 0.000128152;
   DATA[1260,39] := 1.0;
   DATA[1261,0] := 2.540435;
   DATA[1261,1] := 783.3673;
   DATA[1261,2] := 2.0;
   DATA[1261,3] := 1.0;
   DATA[1261,4] := 262.5288;
   DATA[1261,5] := 8.464369;
   DATA[1261,6] := 317.4827;
   DATA[1261,8] := 1.0;
   DATA[1261,9] := 1.0;
   DATA[1261,10] := 1.0;
   DATA[1261,11] := 2.010372;
   DATA[1261,13] := 1010.959;
   DATA[1261,14] := 1.0;
   DATA[1261,15] := 1.0;
   DATA[1261,16] := 1.0;
   DATA[1261,17] := 1.0;
   DATA[1261,18] := 1.0;
   DATA[1261,19] := 1.0;
   DATA[1261,20] := 148.808;
   DATA[1261,21] := 154.14;
   DATA[1261,22] := 1.715952;
   DATA[1261,23] := 821.7124;
   DATA[1261,24] := 2.0;
   DATA[1261,25] := 2.0;
   DATA[1261,26] := 7.87798;
   DATA[1261,27] := 142.9377;
   DATA[1261,28] := 263.0095;
   DATA[1261,29] := 12.15073;
   DATA[1261,30] := 1.725583;
   DATA[1261,31] := 1.280646;
   DATA[1261,32] := 0.7352687;
   DATA[1261,33] := 0.3082983;
   DATA[1261,34] := 2.0;
   DATA[1261,35] := 250.1762;
   DATA[1261,36] := 1.69801;
   DATA[1261,37] := 189.1022;
   DATA[1261,38] := 0.000128152;
   DATA[1261,39] := 1.0;
   DATA[1262,0] := 2.542036;
   DATA[1262,1] := 783.6421;
   DATA[1262,2] := 2.0;
   DATA[1262,3] := 1.0;
   DATA[1262,4] := 262.5288;
   DATA[1262,5] := 8.464369;
   DATA[1262,6] := 317.4827;
   DATA[1262,8] := 1.0;
   DATA[1262,9] := 1.0;
   DATA[1262,10] := 1.0;
   DATA[1262,11] := 2.010372;
   DATA[1262,13] := 1011.119;
   DATA[1262,14] := 1.0;
   DATA[1262,15] := 1.0;
   DATA[1262,16] := 1.0;
   DATA[1262,17] := 1.0;
   DATA[1262,18] := 1.0;
   DATA[1262,19] := 1.0;
   DATA[1262,20] := 148.808;
   DATA[1262,21] := 154.14;
   DATA[1262,22] := 1.715952;
   DATA[1262,23] := 821.4048;
   DATA[1262,24] := 2.0;
   DATA[1262,25] := 2.0;
   DATA[1262,26] := 7.87798;
   DATA[1262,27] := 142.9377;
   DATA[1262,28] := 263.0095;
   DATA[1262,29] := 12.15073;
   DATA[1262,30] := 1.725455;
   DATA[1262,31] := 1.270911;
   DATA[1262,32] := 0.7352687;
   DATA[1262,33] := 0.3082983;
   DATA[1262,34] := 2.0;
   DATA[1262,35] := 250.1762;
   DATA[1262,36] := 1.69801;
   DATA[1262,37] := 189.1022;
   DATA[1262,38] := 0.000128152;
   DATA[1262,39] := 1.0;
   DATA[1263,0] := 2.544278;
   DATA[1263,1] := 784.2308;
   DATA[1263,2] := 2.0;
   DATA[1263,3] := 1.0;
   DATA[1263,4] := 262.5288;
   DATA[1263,5] := 8.464369;
   DATA[1263,6] := 317.4827;
   DATA[1263,8] := 1.0;
   DATA[1263,9] := 1.0;
   DATA[1263,10] := 1.0;
   DATA[1263,11] := 2.010372;
   DATA[1263,13] := 1011.039;
   DATA[1263,14] := 1.0;
   DATA[1263,15] := 1.0;
   DATA[1263,16] := 1.0;
   DATA[1263,17] := 1.0;
   DATA[1263,18] := 1.0;
   DATA[1263,19] := 1.0;
   DATA[1263,20] := 148.808;
   DATA[1263,21] := 154.14;
   DATA[1263,22] := 1.715952;
   DATA[1263,23] := 821.5586;
   DATA[1263,24] := 2.0;
   DATA[1263,25] := 2.0;
   DATA[1263,26] := 7.87798;
   DATA[1263,27] := 142.9377;
   DATA[1263,28] := 263.0095;
   DATA[1263,29] := 12.15073;
   DATA[1263,30] := 1.725455;
   DATA[1263,31] := 1.257077;
   DATA[1263,32] := 0.7352687;
   DATA[1263,33] := 0.3082983;
   DATA[1263,34] := 2.0;
   DATA[1263,35] := 250.1762;
   DATA[1263,36] := 1.69801;
   DATA[1263,37] := 188.958;
   DATA[1263,38] := 0.000128152;
   DATA[1263,39] := 1.0;
   DATA[1264,0] := 2.545559;
   DATA[1264,1] := 784.7411;
   DATA[1264,2] := 2.0;
   DATA[1264,3] := 1.0;
   DATA[1264,4] := 262.5288;
   DATA[1264,5] := 8.464369;
   DATA[1264,6] := 317.4827;
   DATA[1264,8] := 1.0;
   DATA[1264,9] := 1.0;
   DATA[1264,10] := 1.0;
   DATA[1264,11] := 2.010372;
   DATA[1264,13] := 1010.879;
   DATA[1264,14] := 1.0;
   DATA[1264,15] := 1.0;
   DATA[1264,16] := 1.0;
   DATA[1264,17] := 1.0;
   DATA[1264,18] := 1.0;
   DATA[1264,19] := 1.0;
   DATA[1264,20] := 148.808;
   DATA[1264,21] := 154.14;
   DATA[1264,22] := 1.715952;
   DATA[1264,23] := 821.0203;
   DATA[1264,24] := 2.0;
   DATA[1264,25] := 2.0;
   DATA[1264,26] := 7.87798;
   DATA[1264,27] := 142.9377;
   DATA[1264,28] := 263.0095;
   DATA[1264,29] := 12.11228;
   DATA[1264,30] := 1.726609;
   DATA[1264,31] := 1.259511;
   DATA[1264,32] := 0.7352687;
   DATA[1264,33] := 0.3082983;
   DATA[1264,34] := 2.0;
   DATA[1264,35] := 250.1762;
   DATA[1264,36] := 1.681991;
   DATA[1264,37] := 188.958;
   DATA[1264,38] := 0.000128152;
   DATA[1264,39] := 1.0;
   DATA[1265,0] := 2.547161;
   DATA[1265,1] := 785.0159;
   DATA[1265,2] := 2.0;
   DATA[1265,3] := 1.0;
   DATA[1265,4] := 262.5288;
   DATA[1265,5] := 8.464369;
   DATA[1265,6] := 317.4827;
   DATA[1265,8] := 1.0;
   DATA[1265,9] := 1.0;
   DATA[1265,10] := 1.0;
   DATA[1265,11] := 2.010372;
   DATA[1265,13] := 1010.839;
   DATA[1265,14] := 1.0;
   DATA[1265,15] := 1.0;
   DATA[1265,16] := 1.0;
   DATA[1265,17] := 1.0;
   DATA[1265,18] := 1.0;
   DATA[1265,19] := 1.0;
   DATA[1265,20] := 148.808;
   DATA[1265,21] := 154.14;
   DATA[1265,22] := 1.715952;
   DATA[1265,23] := 820.5204;
   DATA[1265,24] := 2.0;
   DATA[1265,25] := 2.0;
   DATA[1265,26] := 7.87798;
   DATA[1265,27] := 142.9377;
   DATA[1265,28] := 263.0095;
   DATA[1265,29] := 12.11228;
   DATA[1265,30] := 1.726865;
   DATA[1265,31] := 1.261816;
   DATA[1265,32] := 0.7352687;
   DATA[1265,33] := 0.3082983;
   DATA[1265,34] := 2.0;
   DATA[1265,35] := 250.1762;
   DATA[1265,36] := 1.681991;
   DATA[1265,37] := 188.958;
   DATA[1265,38] := 0.000128152;
   DATA[1265,39] := 1.0;
   DATA[1266,0] := 2.550684;
   DATA[1266,1] := 785.6047;
   DATA[1266,2] := 2.0;
   DATA[1266,3] := 1.0;
   DATA[1266,4] := 262.5288;
   DATA[1266,5] := 8.464369;
   DATA[1266,6] := 317.4827;
   DATA[1266,8] := 1.0;
   DATA[1266,9] := 1.0;
   DATA[1266,10] := 1.0;
   DATA[1266,11] := 2.010372;
   DATA[1266,13] := 1010.839;
   DATA[1266,14] := 1.0;
   DATA[1266,15] := 1.0;
   DATA[1266,16] := 1.0;
   DATA[1266,17] := 1.0;
   DATA[1266,18] := 1.0;
   DATA[1266,19] := 1.0;
   DATA[1266,20] := 148.808;
   DATA[1266,21] := 154.14;
   DATA[1266,22] := 1.715952;
   DATA[1266,23] := 820.2512;
   DATA[1266,24] := 2.0;
   DATA[1266,25] := 2.0;
   DATA[1266,26] := 7.87798;
   DATA[1266,27] := 142.9377;
   DATA[1266,28] := 263.0095;
   DATA[1266,29] := 12.11228;
   DATA[1266,30] := 1.726865;
   DATA[1266,31] := 1.257077;
   DATA[1266,32] := 0.7352687;
   DATA[1266,33] := 0.3099638;
   DATA[1266,34] := 2.0;
   DATA[1266,35] := 250.1762;
   DATA[1266,36] := 1.681991;
   DATA[1266,37] := 188.958;
   DATA[1266,38] := 0.000128152;
   DATA[1266,39] := 1.0;
   DATA[1267,0] := 2.550684;
   DATA[1267,1] := 786.272;
   DATA[1267,2] := 2.0;
   DATA[1267,3] := 1.0;
   DATA[1267,4] := 262.5288;
   DATA[1267,5] := 8.464369;
   DATA[1267,6] := 317.4827;
   DATA[1267,8] := 1.0;
   DATA[1267,9] := 1.0;
   DATA[1267,10] := 1.0;
   DATA[1267,11] := 2.010372;
   DATA[1267,13] := 1010.959;
   DATA[1267,14] := 1.0;
   DATA[1267,15] := 1.0;
   DATA[1267,16] := 1.0;
   DATA[1267,17] := 1.0;
   DATA[1267,18] := 1.0;
   DATA[1267,19] := 1.0;
   DATA[1267,20] := 148.808;
   DATA[1267,21] := 154.1656;
   DATA[1267,22] := 1.715952;
   DATA[1267,23] := 819.6744;
   DATA[1267,24] := 2.0;
   DATA[1267,25] := 2.0;
   DATA[1267,26] := 7.87798;
   DATA[1267,27] := 142.9377;
   DATA[1267,28] := 263.0095;
   DATA[1267,29] := 12.11228;
   DATA[1267,30] := 1.725455;
   DATA[1267,31] := 1.267068;
   DATA[1267,32] := 0.7352687;
   DATA[1267,33] := 0.3104122;
   DATA[1267,34] := 2.0;
   DATA[1267,35] := 250.0961;
   DATA[1267,36] := 1.681991;
   DATA[1267,37] := 188.958;
   DATA[1267,38] := 0.000128152;
   DATA[1267,39] := 1.0;
   DATA[1268,0] := 2.550684;
   DATA[1268,1] := 786.743;
   DATA[1268,2] := 2.0;
   DATA[1268,3] := 1.0;
   DATA[1268,4] := 262.5288;
   DATA[1268,5] := 8.464369;
   DATA[1268,6] := 317.4827;
   DATA[1268,8] := 1.0;
   DATA[1268,9] := 1.0;
   DATA[1268,10] := 1.0;
   DATA[1268,11] := 2.010372;
   DATA[1268,13] := 1011.079;
   DATA[1268,14] := 1.0;
   DATA[1268,15] := 1.0;
   DATA[1268,16] := 1.0;
   DATA[1268,17] := 1.0;
   DATA[1268,18] := 1.0;
   DATA[1268,19] := 1.0;
   DATA[1268,20] := 148.808;
   DATA[1268,21] := 154.1656;
   DATA[1268,22] := 1.714798;
   DATA[1268,23] := 819.5975;
   DATA[1268,24] := 2.0;
   DATA[1268,25] := 2.0;
   DATA[1268,26] := 7.87798;
   DATA[1268,27] := 142.9377;
   DATA[1268,28] := 263.0095;
   DATA[1268,29] := 12.11228;
   DATA[1268,30] := 1.723789;
   DATA[1268,31] := 1.271551;
   DATA[1268,32] := 0.7352687;
   DATA[1268,33] := 0.3104122;
   DATA[1268,34] := 2.0;
   DATA[1268,35] := 250.0961;
   DATA[1268,36] := 1.681991;
   DATA[1268,37] := 188.958;
   DATA[1268,38] := 0.000128152;
   DATA[1268,39] := 1.0;
   DATA[1269,0] := 2.545559;
   DATA[1269,1] := 787.0571;
   DATA[1269,2] := 2.0;
   DATA[1269,3] := 1.0;
   DATA[1269,4] := 262.5288;
   DATA[1269,5] := 8.464369;
   DATA[1269,6] := 317.4827;
   DATA[1269,8] := 1.0;
   DATA[1269,9] := 1.0;
   DATA[1269,10] := 1.0;
   DATA[1269,11] := 2.010372;
   DATA[1269,13] := 1011.079;
   DATA[1269,14] := 1.0;
   DATA[1269,15] := 1.0;
   DATA[1269,16] := 1.0;
   DATA[1269,17] := 1.0;
   DATA[1269,18] := 1.0;
   DATA[1269,19] := 1.0;
   DATA[1269,20] := 148.808;
   DATA[1269,21] := 154.1656;
   DATA[1269,22] := 1.713261;
   DATA[1269,23] := 819.2899;
   DATA[1269,24] := 2.0;
   DATA[1269,25] := 2.0;
   DATA[1269,26] := 7.87798;
   DATA[1269,27] := 142.9377;
   DATA[1269,28] := 263.0095;
   DATA[1269,29] := 12.11228;
   DATA[1269,30] := 1.723789;
   DATA[1269,31] := 1.277187;
   DATA[1269,32] := 0.7352687;
   DATA[1269,33] := 0.3084265;
   DATA[1269,34] := 2.0;
   DATA[1269,35] := 250.0961;
   DATA[1269,36] := 1.681991;
   DATA[1269,37] := 188.958;
   DATA[1269,38] := 0.000128152;
   DATA[1269,39] := 1.0;
   DATA[1270,0] := 2.543317;
   DATA[1270,1] := 787.9598;
   DATA[1270,2] := 2.0;
   DATA[1270,3] := 1.0;
   DATA[1270,4] := 262.5288;
   DATA[1270,5] := 8.464369;
   DATA[1270,6] := 317.4827;
   DATA[1270,8] := 1.0;
   DATA[1270,9] := 1.0;
   DATA[1270,10] := 1.0;
   DATA[1270,11] := 1.997567;
   DATA[1270,12] := 0.000256221;
   DATA[1270,13] := 1011.039;
   DATA[1270,14] := 1.0;
   DATA[1270,15] := 1.0;
   DATA[1270,16] := 1.0;
   DATA[1270,17] := 1.0;
   DATA[1270,18] := 1.0;
   DATA[1270,19] := 1.0;
   DATA[1270,20] := 148.808;
   DATA[1270,21] := 154.1656;
   DATA[1270,22] := 1.713261;
   DATA[1270,23] := 819.0977;
   DATA[1270,24] := 2.0;
   DATA[1270,25] := 2.0;
   DATA[1270,26] := 7.87798;
   DATA[1270,27] := 142.9377;
   DATA[1270,28] := 263.0095;
   DATA[1270,29] := 12.11228;
   DATA[1270,30] := 1.723789;
   DATA[1270,31] := 1.281158;
   DATA[1270,32] := 0.7352687;
   DATA[1270,33] := 0.3082983;
   DATA[1270,34] := 2.0;
   DATA[1270,35] := 250.0961;
   DATA[1270,36] := 1.681991;
   DATA[1270,37] := 188.958;
   DATA[1270,38] := 0.000128152;
   DATA[1270,39] := 1.0;
   DATA[1271,0] := 2.541716;
   DATA[1271,1] := 788.6271;
   DATA[1271,2] := 2.0;
   DATA[1271,3] := 1.0;
   DATA[1271,4] := 262.5288;
   DATA[1271,5] := 8.464369;
   DATA[1271,6] := 317.4827;
   DATA[1271,8] := 1.0;
   DATA[1271,9] := 1.0;
   DATA[1271,10] := 1.0;
   DATA[1271,11] := 1.997567;
   DATA[1271,12] := 0.000256221;
   DATA[1271,13] := 1010.919;
   DATA[1271,14] := 1.0;
   DATA[1271,15] := 1.0;
   DATA[1271,16] := 1.0;
   DATA[1271,17] := 1.0;
   DATA[1271,18] := 1.0;
   DATA[1271,19] := 1.0;
   DATA[1271,20] := 148.808;
   DATA[1271,21] := 154.1656;
   DATA[1271,22] := 1.713261;
   DATA[1271,23] := 818.79;
   DATA[1271,24] := 2.0;
   DATA[1271,25] := 2.0;
   DATA[1271,26] := 7.87798;
   DATA[1271,27] := 142.9377;
   DATA[1271,28] := 263.0095;
   DATA[1271,29] := 12.11228;
   DATA[1271,30] := 1.723789;
   DATA[1271,31] := 1.27296;
   DATA[1271,32] := 0.7352687;
   DATA[1271,33] := 0.3082983;
   DATA[1271,34] := 2.0;
   DATA[1271,35] := 250.0961;
   DATA[1271,36] := 1.681991;
   DATA[1271,37] := 188.8618;
   DATA[1271,38] := 0.000128152;
   DATA[1271,39] := 1.0;
   DATA[1272,0] := 2.539474;
   DATA[1272,1] := 789.2159;
   DATA[1272,2] := 2.0;
   DATA[1272,3] := 1.0;
   DATA[1272,4] := 262.5288;
   DATA[1272,5] := 8.464369;
   DATA[1272,6] := 317.4827;
   DATA[1272,8] := 1.0;
   DATA[1272,9] := 1.0;
   DATA[1272,10] := 1.0;
   DATA[1272,11] := 1.997567;
   DATA[1272,12] := 0.000256221;
   DATA[1272,13] := 1010.758;
   DATA[1272,14] := 1.0;
   DATA[1272,15] := 1.0;
   DATA[1272,16] := 1.0;
   DATA[1272,17] := 1.0;
   DATA[1272,18] := 1.0;
   DATA[1272,19] := 1.0;
   DATA[1272,20] := 148.808;
   DATA[1272,21] := 154.1656;
   DATA[1272,22] := 1.71608;
   DATA[1272,23] := 818.2517;
   DATA[1272,24] := 2.0;
   DATA[1272,25] := 2.0;
   DATA[1272,26] := 7.87798;
   DATA[1272,27] := 142.8352;
   DATA[1272,28] := 263.0095;
   DATA[1272,29] := 12.11228;
   DATA[1272,30] := 1.723789;
   DATA[1272,31] := 1.271039;
   DATA[1272,32] := 0.7352687;
   DATA[1272,33] := 0.3082983;
   DATA[1272,34] := 2.0;
   DATA[1272,35] := 250.0961;
   DATA[1272,36] := 1.762086;
   DATA[1272,37] := 188.8618;
   DATA[1272,38] := 0.000128152;
   DATA[1272,39] := 1.0;
   DATA[1273,0] := 2.539474;
   DATA[1273,1] := 789.4907;
   DATA[1273,2] := 2.0;
   DATA[1273,3] := 1.0;
   DATA[1273,4] := 262.5288;
   DATA[1273,5] := 8.464369;
   DATA[1273,6] := 317.4827;
   DATA[1273,8] := 1.0;
   DATA[1273,9] := 1.0;
   DATA[1273,10] := 1.0;
   DATA[1273,11] := 1.997567;
   DATA[1273,12] := 0.000256221;
   DATA[1273,13] := 1010.879;
   DATA[1273,14] := 1.0;
   DATA[1273,15] := 1.0;
   DATA[1273,16] := 1.0;
   DATA[1273,17] := 1.0;
   DATA[1273,18] := 1.0;
   DATA[1273,19] := 1.0;
   DATA[1273,20] := 148.808;
   DATA[1273,21] := 154.1656;
   DATA[1273,22] := 1.71608;
   DATA[1273,23] := 817.8672;
   DATA[1273,24] := 2.0;
   DATA[1273,25] := 2.0;
   DATA[1273,26] := 7.87798;
   DATA[1273,27] := 142.707;
   DATA[1273,28] := 263.0095;
   DATA[1273,29] := 12.11228;
   DATA[1273,30] := 1.723789;
   DATA[1273,31] := 1.272192;
   DATA[1273,32] := 0.7352687;
   DATA[1273,33] := 0.3082983;
   DATA[1273,34] := 2.0;
   DATA[1273,35] := 250.0961;
   DATA[1273,36] := 1.762086;
   DATA[1273,37] := 188.8618;
   DATA[1273,38] := 0.000128152;
   DATA[1273,39] := 1.0;
   DATA[1274,0] := 2.548762;
   DATA[1274,1] := 790.0403;
   DATA[1274,2] := 2.0;
   DATA[1274,3] := 1.0;
   DATA[1274,4] := 262.5288;
   DATA[1274,5] := 8.464369;
   DATA[1274,6] := 317.4827;
   DATA[1274,8] := 1.0;
   DATA[1274,9] := 1.0;
   DATA[1274,10] := 1.0;
   DATA[1274,11] := 1.997567;
   DATA[1274,12] := 0.000256221;
   DATA[1274,13] := 1010.758;
   DATA[1274,14] := 1.0;
   DATA[1274,15] := 1.0;
   DATA[1274,16] := 1.0;
   DATA[1274,17] := 1.0;
   DATA[1274,18] := 1.0;
   DATA[1274,19] := 1.0;
   DATA[1274,20] := 148.808;
   DATA[1274,21] := 154.1656;
   DATA[1274,22] := 1.71608;
   DATA[1274,23] := 817.0598;
   DATA[1274,24] := 2.0;
   DATA[1274,25] := 2.0;
   DATA[1274,26] := 7.87798;
   DATA[1274,27] := 142.707;
   DATA[1274,28] := 263.0095;
   DATA[1274,29] := 12.11228;
   DATA[1274,30] := 1.723789;
   DATA[1274,31] := 1.289612;
   DATA[1274,32] := 0.7352687;
   DATA[1274,33] := 0.3082983;
   DATA[1274,34] := 2.0;
   DATA[1274,35] := 250.0961;
   DATA[1274,36] := 1.762086;
   DATA[1274,37] := 188.8618;
   DATA[1274,38] := 0.000128152;
   DATA[1274,39] := 1.0;
   DATA[1275,0] := 2.548762;
   DATA[1275,1] := 790.0403;
   DATA[1275,2] := 2.0;
   DATA[1275,3] := 1.0;
   DATA[1275,4] := 262.5288;
   DATA[1275,5] := 8.464369;
   DATA[1275,6] := 317.4827;
   DATA[1275,8] := 1.0;
   DATA[1275,9] := 1.0;
   DATA[1275,10] := 1.0;
   DATA[1275,11] := 1.997567;
   DATA[1275,12] := 0.000256221;
   DATA[1275,13] := 1010.758;
   DATA[1275,14] := 1.0;
   DATA[1275,15] := 1.0;
   DATA[1275,16] := 1.0;
   DATA[1275,17] := 1.0;
   DATA[1275,18] := 1.0;
   DATA[1275,19] := 1.0;
   DATA[1275,20] := 148.808;
   DATA[1275,21] := 154.1656;
   DATA[1275,22] := 1.71608;
   DATA[1275,23] := 817.0598;
   DATA[1275,24] := 2.0;
   DATA[1275,25] := 2.0;
   DATA[1275,26] := 7.87798;
   DATA[1275,27] := 142.707;
   DATA[1275,28] := 263.0095;
   DATA[1275,29] := 12.11228;
   DATA[1275,30] := 1.723789;
   DATA[1275,31] := 1.289612;
   DATA[1275,32] := 0.7352687;
   DATA[1275,33] := 0.3082983;
   DATA[1275,34] := 2.0;
   DATA[1275,35] := 250.0961;
   DATA[1275,36] := 1.762086;
   DATA[1275,37] := 188.8618;
   DATA[1275,38] := 0.000128152;
   DATA[1275,39] := 1.0;
   DATA[1276,0] := 2.550364;
   DATA[1276,1] := 790.7076;
   DATA[1276,2] := 2.0;
   DATA[1276,3] := 1.0;
   DATA[1276,4] := 262.5288;
   DATA[1276,5] := 8.464369;
   DATA[1276,6] := 317.4827;
   DATA[1276,8] := 1.0;
   DATA[1276,9] := 1.0;
   DATA[1276,10] := 1.0;
   DATA[1276,11] := 1.997567;
   DATA[1276,12] := 0.000256221;
   DATA[1276,13] := 1011.039;
   DATA[1276,14] := 1.0;
   DATA[1276,15] := 1.0;
   DATA[1276,16] := 1.0;
   DATA[1276,17] := 1.0;
   DATA[1276,18] := 1.0;
   DATA[1276,19] := 1.0;
   DATA[1276,20] := 148.808;
   DATA[1276,21] := 154.1656;
   DATA[1276,22] := 1.71608;
   DATA[1276,23] := 816.9444;
   DATA[1276,24] := 2.0;
   DATA[1276,25] := 2.0;
   DATA[1276,26] := 7.87798;
   DATA[1276,27] := 142.707;
   DATA[1276,28] := 263.0095;
   DATA[1276,29] := 12.11228;
   DATA[1276,30] := 1.723789;
   DATA[1276,31] := 1.292046;
   DATA[1276,32] := 0.7352687;
   DATA[1276,33] := 0.3082983;
   DATA[1276,34] := 2.0;
   DATA[1276,35] := 250.0961;
   DATA[1276,36] := 1.762086;
   DATA[1276,37] := 188.958;
   DATA[1276,38] := 0.000128152;
   DATA[1276,39] := 1.0;
   DATA[1277,0] := 2.551645;
   DATA[1277,1] := 791.2963;
   DATA[1277,2] := 2.0;
   DATA[1277,3] := 1.0;
   DATA[1277,4] := 262.5288;
   DATA[1277,5] := 8.464369;
   DATA[1277,6] := 317.6878;
   DATA[1277,8] := 1.0;
   DATA[1277,9] := 1.0;
   DATA[1277,10] := 1.0;
   DATA[1277,11] := 1.997567;
   DATA[1277,12] := 0.000256221;
   DATA[1277,13] := 1010.959;
   DATA[1277,14] := 1.0;
   DATA[1277,15] := 1.0;
   DATA[1277,16] := 1.0;
   DATA[1277,17] := 1.0;
   DATA[1277,18] := 1.0;
   DATA[1277,19] := 1.0;
   DATA[1277,20] := 148.808;
   DATA[1277,21] := 154.1656;
   DATA[1277,22] := 1.71608;
   DATA[1277,23] := 816.2907;
   DATA[1277,24] := 2.0;
   DATA[1277,25] := 2.0;
   DATA[1277,26] := 7.87798;
   DATA[1277,27] := 142.707;
   DATA[1277,28] := 263.0095;
   DATA[1277,29] := 12.11228;
   DATA[1277,30] := 1.723789;
   DATA[1277,31] := 1.287434;
   DATA[1277,32] := 0.7352687;
   DATA[1277,33] := 0.3082983;
   DATA[1277,34] := 2.0;
   DATA[1277,35] := 250.0961;
   DATA[1277,36] := 1.665972;
   DATA[1277,37] := 188.958;
   DATA[1277,38] := 0.000128152;
   DATA[1277,39] := 1.0;
   DATA[1278,0] := 2.552285;
   DATA[1278,1] := 791.2963;
   DATA[1278,2] := 2.0;
   DATA[1278,3] := 1.0;
   DATA[1278,4] := 262.5288;
   DATA[1278,5] := 8.464369;
   DATA[1278,6] := 317.6878;
   DATA[1278,8] := 1.0;
   DATA[1278,9] := 1.0;
   DATA[1278,10] := 1.0;
   DATA[1278,11] := 2.013573;
   DATA[1278,12] := 0.000256221;
   DATA[1278,13] := 1011.359;
   DATA[1278,14] := 1.0;
   DATA[1278,15] := 1.0;
   DATA[1278,16] := 1.0;
   DATA[1278,17] := 1.0;
   DATA[1278,18] := 1.0;
   DATA[1278,19] := 1.0;
   DATA[1278,20] := 148.808;
   DATA[1278,21] := 154.1656;
   DATA[1278,22] := 1.71608;
   DATA[1278,23] := 815.8293;
   DATA[1278,24] := 2.0;
   DATA[1278,25] := 2.0;
   DATA[1278,26] := 7.87798;
   DATA[1278,27] := 142.8095;
   DATA[1278,28] := 263.0095;
   DATA[1278,29] := 12.11228;
   DATA[1278,30] := 1.723789;
   DATA[1278,31] := 1.287434;
   DATA[1278,32] := 0.7352687;
   DATA[1278,33] := 0.3082983;
   DATA[1278,34] := 2.0;
   DATA[1278,35] := 250.0961;
   DATA[1278,36] := 1.665972;
   DATA[1278,37] := 188.958;
   DATA[1278,38] := 0.000128152;
   DATA[1278,39] := 1.0;
   DATA[1279,0] := 2.555488;
   DATA[1279,1] := 791.6889;
   DATA[1279,2] := 2.0;
   DATA[1279,3] := 1.0;
   DATA[1279,4] := 262.5288;
   DATA[1279,5] := 8.464369;
   DATA[1279,6] := 317.6878;
   DATA[1279,8] := 1.0;
   DATA[1279,9] := 1.0;
   DATA[1279,10] := 1.0;
   DATA[1279,11] := 2.013573;
   DATA[1279,12] := 0.000256221;
   DATA[1279,13] := 1011.039;
   DATA[1279,14] := 1.0;
   DATA[1279,15] := 1.0;
   DATA[1279,16] := 1.0;
   DATA[1279,17] := 1.0;
   DATA[1279,18] := 1.0;
   DATA[1279,19] := 1.0;
   DATA[1279,20] := 148.808;
   DATA[1279,21] := 154.1143;
   DATA[1279,22] := 1.71608;
   DATA[1279,23] := 815.4448;
   DATA[1279,24] := 2.0;
   DATA[1279,25] := 2.0;
   DATA[1279,26] := 7.87798;
   DATA[1279,27] := 142.8095;
   DATA[1279,28] := 263.0095;
   DATA[1279,29] := 12.11228;
   DATA[1279,30] := 1.723789;
   DATA[1279,31] := 1.282823;
   DATA[1279,32] := 0.7352687;
   DATA[1279,33] := 0.3082983;
   DATA[1279,34] := 2.0;
   DATA[1279,35] := 250.0961;
   DATA[1279,36] := 1.665972;
   DATA[1279,37] := 188.958;
   DATA[1279,38] := 0.000128152;
   DATA[1279,39] := 1.0;
   DATA[1280,0] := 2.555488;
   DATA[1280,1] := 792.1599;
   DATA[1280,2] := 2.0;
   DATA[1280,3] := 1.0;
   DATA[1280,4] := 262.5288;
   DATA[1280,5] := 8.464369;
   DATA[1280,6] := 317.6878;
   DATA[1280,8] := 1.0;
   DATA[1280,9] := 1.0;
   DATA[1280,10] := 1.0;
   DATA[1280,11] := 2.013573;
   DATA[1280,12] := 0.000256221;
   DATA[1280,13] := 1010.558;
   DATA[1280,14] := 1.0;
   DATA[1280,15] := 1.0;
   DATA[1280,16] := 1.0;
   DATA[1280,17] := 1.0;
   DATA[1280,18] := 1.0;
   DATA[1280,19] := 1.0;
   DATA[1280,20] := 148.808;
   DATA[1280,21] := 153.8836;
   DATA[1280,22] := 1.71608;
   DATA[1280,23] := 815.0218;
   DATA[1280,24] := 2.0;
   DATA[1280,25] := 2.0;
   DATA[1280,26] := 7.87798;
   DATA[1280,27] := 142.8095;
   DATA[1280,28] := 263.0095;
   DATA[1280,29] := 12.11228;
   DATA[1280,30] := 1.723789;
   DATA[1280,31] := 1.282183;
   DATA[1280,32] := 0.7352687;
   DATA[1280,33] := 0.3082983;
   DATA[1280,34] := 2.0;
   DATA[1280,35] := 250.0961;
   DATA[1280,36] := 1.665972;
   DATA[1280,37] := 188.958;
   DATA[1280,38] := 0.000128152;
   DATA[1280,39] := 1.0;
   DATA[1281,0] := 2.548121;
   DATA[1281,1] := 792.8272;
   DATA[1281,2] := 2.0;
   DATA[1281,3] := 1.0;
   DATA[1281,4] := 262.5288;
   DATA[1281,5] := 8.464369;
   DATA[1281,6] := 317.6878;
   DATA[1281,8] := 1.0;
   DATA[1281,9] := 1.0;
   DATA[1281,10] := 1.0;
   DATA[1281,11] := 2.013573;
   DATA[1281,12] := 0.000256221;
   DATA[1281,13] := 1010.959;
   DATA[1281,14] := 1.0;
   DATA[1281,15] := 1.0;
   DATA[1281,16] := 1.0;
   DATA[1281,17] := 1.0;
   DATA[1281,18] := 1.0;
   DATA[1281,19] := 1.0;
   DATA[1281,20] := 148.808;
   DATA[1281,21] := 153.8836;
   DATA[1281,22] := 1.71608;
   DATA[1281,23] := 814.5604;
   DATA[1281,24] := 2.0;
   DATA[1281,25] := 2.0;
   DATA[1281,26] := 7.87798;
   DATA[1281,27] := 142.8095;
   DATA[1281,28] := 263.0095;
   DATA[1281,29] := 12.11228;
   DATA[1281,30] := 1.723789;
   DATA[1281,31] := 1.288075;
   DATA[1281,32] := 0.7352687;
   DATA[1281,33] := 0.3099638;
   DATA[1281,34] := 2.0;
   DATA[1281,35] := 249.984;
   DATA[1281,36] := 1.665972;
   DATA[1281,37] := 188.958;
   DATA[1281,38] := 0.000128152;
   DATA[1281,39] := 1.0;
   DATA[1282,0] := 2.54652;
   DATA[1282,1] := 792.9449;
   DATA[1282,2] := 2.0;
   DATA[1282,3] := 1.0;
   DATA[1282,4] := 262.5288;
   DATA[1282,5] := 8.464369;
   DATA[1282,6] := 317.6878;
   DATA[1282,8] := 1.0;
   DATA[1282,9] := 1.0;
   DATA[1282,10] := 1.0;
   DATA[1282,11] := 2.013573;
   DATA[1282,12] := 0.000256221;
   DATA[1282,13] := 1010.758;
   DATA[1282,14] := 1.0;
   DATA[1282,15] := 1.0;
   DATA[1282,16] := 1.0;
   DATA[1282,17] := 1.0;
   DATA[1282,18] := 1.0;
   DATA[1282,19] := 1.0;
   DATA[1282,20] := 148.808;
   DATA[1282,21] := 153.8836;
   DATA[1282,22] := 1.71608;
   DATA[1282,23] := 814.0605;
   DATA[1282,24] := 2.0;
   DATA[1282,25] := 2.0;
   DATA[1282,26] := 7.87798;
   DATA[1282,27] := 142.8095;
   DATA[1282,28] := 263.0095;
   DATA[1282,29] := 12.11228;
   DATA[1282,30] := 1.723789;
   DATA[1282,31] := 1.283079;
   DATA[1282,32] := 0.7352687;
   DATA[1282,33] := 0.3109887;
   DATA[1282,34] := 2.0;
   DATA[1282,35] := 249.6956;
   DATA[1282,36] := 1.665972;
   DATA[1282,37] := 188.6535;
   DATA[1282,38] := 0.000128152;
   DATA[1282,39] := 1.0;
   DATA[1283,0] := 2.539154;
   DATA[1283,1] := 793.1805;
   DATA[1283,2] := 2.0;
   DATA[1283,3] := 1.0;
   DATA[1283,4] := 262.5288;
   DATA[1283,5] := 8.464369;
   DATA[1283,6] := 317.6878;
   DATA[1283,8] := 1.0;
   DATA[1283,9] := 1.0;
   DATA[1283,10] := 1.0;
   DATA[1283,11] := 2.013573;
   DATA[1283,12] := 0.000256221;
   DATA[1283,13] := 1011.239;
   DATA[1283,14] := 1.0;
   DATA[1283,15] := 1.0;
   DATA[1283,16] := 1.0;
   DATA[1283,17] := 1.0;
   DATA[1283,18] := 1.0;
   DATA[1283,19] := 1.0;
   DATA[1283,20] := 148.808;
   DATA[1283,21] := 154.1912;
   DATA[1283,22] := 1.714029;
   DATA[1283,23] := 813.4453;
   DATA[1283,24] := 2.0;
   DATA[1283,25] := 2.0;
   DATA[1283,26] := 7.87798;
   DATA[1283,27] := 142.8352;
   DATA[1283,28] := 263.0095;
   DATA[1283,29] := 12.11228;
   DATA[1283,30] := 1.72302;
   DATA[1283,31] := 1.282311;
   DATA[1283,32] := 0.7353967;
   DATA[1283,33] := 0.3092592;
   DATA[1283,34] := 2.0;
   DATA[1283,35] := 249.6956;
   DATA[1283,36] := 1.665972;
   DATA[1283,37] := 188.6535;
   DATA[1283,38] := 0.000128152;
   DATA[1283,39] := 1.0;
   DATA[1284,0] := 2.534029;
   DATA[1284,1] := 793.1805;
   DATA[1284,2] := 2.0;
   DATA[1284,3] := 1.0;
   DATA[1284,4] := 262.5288;
   DATA[1284,5] := 8.464369;
   DATA[1284,6] := 317.6878;
   DATA[1284,8] := 1.0;
   DATA[1284,9] := 1.0;
   DATA[1284,10] := 1.0;
   DATA[1284,11] := 1.994366;
   DATA[1284,12] := 0.000256221;
   DATA[1284,13] := 1010.879;
   DATA[1284,14] := 1.0;
   DATA[1284,15] := 1.0;
   DATA[1284,16] := 1.0;
   DATA[1284,17] := 1.0;
   DATA[1284,18] := 1.0;
   DATA[1284,19] := 1.0;
   DATA[1284,20] := 148.808;
   DATA[1284,21] := 154.1912;
   DATA[1284,22] := 1.712876;
   DATA[1284,23] := 813.6375;
   DATA[1284,24] := 2.0;
   DATA[1284,25] := 2.0;
   DATA[1284,26] := 7.87798;
   DATA[1284,27] := 143.0403;
   DATA[1284,28] := 263.0095;
   DATA[1284,29] := 12.11228;
   DATA[1284,30] := 1.72161;
   DATA[1284,31] := 1.274497;
   DATA[1284,32] := 0.7371892;
   DATA[1284,33] := 0.3091311;
   DATA[1284,34] := 2.0;
   DATA[1284,35] := 249.6956;
   DATA[1284,36] := 1.665972;
   DATA[1284,37] := 188.6535;
   DATA[1284,38] := 0.000128152;
   DATA[1284,39] := 1.0;
   DATA[1285,0] := 2.534029;
   DATA[1285,1] := 793.1805;
   DATA[1285,2] := 2.0;
   DATA[1285,3] := 1.0;
   DATA[1285,4] := 262.5288;
   DATA[1285,5] := 8.464369;
   DATA[1285,6] := 317.6878;
   DATA[1285,8] := 1.0;
   DATA[1285,9] := 1.0;
   DATA[1285,10] := 1.0;
   DATA[1285,11] := 1.994366;
   DATA[1285,12] := 0.000256221;
   DATA[1285,13] := 1011.279;
   DATA[1285,14] := 1.0;
   DATA[1285,15] := 1.0;
   DATA[1285,16] := 1.0;
   DATA[1285,17] := 1.0;
   DATA[1285,18] := 1.0;
   DATA[1285,19] := 1.0;
   DATA[1285,20] := 148.808;
   DATA[1285,21] := 154.0118;
   DATA[1285,22] := 1.71262;
   DATA[1285,23] := 813.4837;
   DATA[1285,24] := 2.0;
   DATA[1285,25] := 2.0;
   DATA[1285,26] := 7.87798;
   DATA[1285,27] := 143.0403;
   DATA[1285,28] := 263.0095;
   DATA[1285,29] := 12.11228;
   DATA[1285,30] := 1.72161;
   DATA[1285,31] := 1.272064;
   DATA[1285,32] := 0.7378293;
   DATA[1285,33] := 0.3091311;
   DATA[1285,34] := 2.0;
   DATA[1285,35] := 249.6956;
   DATA[1285,36] := 1.665972;
   DATA[1285,37] := 188.6215;
   DATA[1285,38] := 0.000128152;
   DATA[1285,39] := 1.0;
   DATA[1286,0] := 2.532748;
   DATA[1286,1] := 794.2403;
   DATA[1286,2] := 2.0;
   DATA[1286,3] := 1.0;
   DATA[1286,4] := 262.5288;
   DATA[1286,5] := 8.464369;
   DATA[1286,6] := 317.6878;
   DATA[1286,8] := 1.0;
   DATA[1286,9] := 1.0;
   DATA[1286,10] := 1.0;
   DATA[1286,11] := 1.994366;
   DATA[1286,12] := 0.000256221;
   DATA[1286,13] := 1010.919;
   DATA[1286,14] := 1.0;
   DATA[1286,15] := 1.0;
   DATA[1286,16] := 1.0;
   DATA[1286,17] := 1.0;
   DATA[1286,18] := 1.0;
   DATA[1286,19] := 1.0;
   DATA[1286,20] := 148.808;
   DATA[1286,21] := 154.0118;
   DATA[1286,22] := 1.71262;
   DATA[1286,23] := 813.2145;
   DATA[1286,24] := 2.0;
   DATA[1286,25] := 2.0;
   DATA[1286,26] := 7.87798;
   DATA[1286,27] := 143.0403;
   DATA[1286,28] := 263.0095;
   DATA[1286,29] := 12.11228;
   DATA[1286,30] := 1.72161;
   DATA[1286,31] := 1.276803;
   DATA[1286,32] := 0.7378293;
   DATA[1286,33] := 0.3106684;
   DATA[1286,34] := 2.0;
   DATA[1286,35] := 249.6956;
   DATA[1286,36] := 1.665972;
   DATA[1286,37] := 188.6215;
   DATA[1286,38] := 0.000128152;
   DATA[1286,39] := 1.0;
   DATA[1287,0] := 2.532748;
   DATA[1287,1] := 794.7114;
   DATA[1287,2] := 2.0;
   DATA[1287,3] := 1.0;
   DATA[1287,4] := 262.5288;
   DATA[1287,5] := 8.464369;
   DATA[1287,6] := 317.6878;
   DATA[1287,8] := 1.0;
   DATA[1287,9] := 1.0;
   DATA[1287,10] := 1.0;
   DATA[1287,11] := 1.997567;
   DATA[1287,12] := 0.000256221;
   DATA[1287,13] := 1011.119;
   DATA[1287,14] := 1.0;
   DATA[1287,15] := 1.0;
   DATA[1287,16] := 1.0;
   DATA[1287,17] := 1.0;
   DATA[1287,18] := 1.0;
   DATA[1287,19] := 1.0;
   DATA[1287,20] := 148.808;
   DATA[1287,21] := 154.0118;
   DATA[1287,22] := 1.71262;
   DATA[1287,23] := 812.5609;
   DATA[1287,24] := 2.0;
   DATA[1287,25] := 2.0;
   DATA[1287,26] := 7.87798;
   DATA[1287,27] := 143.0403;
   DATA[1287,28] := 263.0095;
   DATA[1287,29] := 12.11228;
   DATA[1287,30] := 1.72161;
   DATA[1287,31] := 1.266428;
   DATA[1287,32] := 0.7378293;
   DATA[1287,33] := 0.3106684;
   DATA[1287,34] := 2.0;
   DATA[1287,35] := 249.6956;
   DATA[1287,36] := 1.665972;
   DATA[1287,37] := 188.6215;
   DATA[1287,38] := 0.000128152;
   DATA[1287,39] := 1.0;
   DATA[1288,0] := 2.539154;
   DATA[1288,1] := 794.9861;
   DATA[1288,2] := 2.0;
   DATA[1288,3] := 1.0;
   DATA[1288,4] := 262.5288;
   DATA[1288,5] := 8.464369;
   DATA[1288,6] := 317.6878;
   DATA[1288,8] := 1.0;
   DATA[1288,9] := 1.0;
   DATA[1288,10] := 1.0;
   DATA[1288,11] := 1.997567;
   DATA[1288,12] := 0.000256221;
   DATA[1288,13] := 1010.919;
   DATA[1288,14] := 1.0;
   DATA[1288,15] := 1.0;
   DATA[1288,16] := 1.0;
   DATA[1288,17] := 1.0;
   DATA[1288,18] := 1.0;
   DATA[1288,19] := 1.0;
   DATA[1288,20] := 148.808;
   DATA[1288,21] := 154.0118;
   DATA[1288,22] := 1.71262;
   DATA[1288,23] := 812.2917;
   DATA[1288,24] := 2.0;
   DATA[1288,25] := 2.0;
   DATA[1288,26] := 7.87798;
   DATA[1288,27] := 143.0403;
   DATA[1288,28] := 263.0095;
   DATA[1288,29] := 12.11228;
   DATA[1288,30] := 1.72161;
   DATA[1288,31] := 1.262073;
   DATA[1288,32] := 0.7378293;
   DATA[1288,33] := 0.3084265;
   DATA[1288,34] := 2.0;
   DATA[1288,35] := 249.6956;
   DATA[1288,36] := 1.665972;
   DATA[1288,37] := 188.6215;
   DATA[1288,38] := 0.000128152;
   DATA[1288,39] := 1.0;
   DATA[1289,0] := 2.544919;
   DATA[1289,1] := 795.7319;
   DATA[1289,2] := 2.0;
   DATA[1289,3] := 1.0;
   DATA[1289,4] := 262.5288;
   DATA[1289,5] := 8.464369;
   DATA[1289,6] := 317.6878;
   DATA[1289,8] := 1.0;
   DATA[1289,9] := 1.0;
   DATA[1289,10] := 1.0;
   DATA[1289,11] := 1.997567;
   DATA[1289,12] := 0.000256221;
   DATA[1289,13] := 1011.079;
   DATA[1289,14] := 1.0;
   DATA[1289,15] := 1.0;
   DATA[1289,16] := 1.0;
   DATA[1289,17] := 1.0;
   DATA[1289,18] := 1.0;
   DATA[1289,19] := 1.0;
   DATA[1289,20] := 148.808;
   DATA[1289,21] := 154.0118;
   DATA[1289,22] := 1.714798;
   DATA[1289,23] := 811.9841;
   DATA[1289,24] := 2.0;
   DATA[1289,25] := 2.0;
   DATA[1289,26] := 7.87798;
   DATA[1289,27] := 143.0403;
   DATA[1289,28] := 263.0095;
   DATA[1289,29] := 12.26609;
   DATA[1289,30] := 1.72161;
   DATA[1289,31] := 1.271295;
   DATA[1289,32] := 0.7378293;
   DATA[1289,33] := 0.3082983;
   DATA[1289,34] := 2.0;
   DATA[1289,35] := 249.984;
   DATA[1289,36] := 1.665972;
   DATA[1289,37] := 188.7977;
   DATA[1289,38] := 0.000128152;
   DATA[1289,39] := 1.0;
   DATA[1290,0] := 2.545239;
   DATA[1290,1] := 796.1245;
   DATA[1290,2] := 2.0;
   DATA[1290,3] := 1.0;
   DATA[1290,4] := 262.5609;
   DATA[1290,5] := 8.464369;
   DATA[1290,6] := 317.6878;
   DATA[1290,8] := 1.0;
   DATA[1290,9] := 1.0;
   DATA[1290,10] := 1.0;
   DATA[1290,11] := 1.997567;
   DATA[1290,12] := 0.000256221;
   DATA[1290,13] := 1010.959;
   DATA[1290,14] := 1.0;
   DATA[1290,15] := 1.0;
   DATA[1290,16] := 1.0;
   DATA[1290,17] := 1.0;
   DATA[1290,18] := 1.0;
   DATA[1290,19] := 1.0;
   DATA[1290,20] := 148.808;
   DATA[1290,21] := 154.0118;
   DATA[1290,22] := 1.714798;
   DATA[1290,23] := 811.7919;
   DATA[1290,24] := 2.0;
   DATA[1290,25] := 2.0;
   DATA[1290,26] := 7.87798;
   DATA[1290,27] := 143.0403;
   DATA[1290,28] := 263.0095;
   DATA[1290,29] := 12.26609;
   DATA[1290,30] := 1.723789;
   DATA[1290,31] := 1.279365;
   DATA[1290,32] := 0.7378293;
   DATA[1290,33] := 0.3082983;
   DATA[1290,34] := 2.0;
   DATA[1290,35] := 249.984;
   DATA[1290,36] := 1.730048;
   DATA[1290,37] := 188.8939;
   DATA[1290,38] := 0.000128152;
   DATA[1290,39] := 1.0;
   DATA[1291,0] := 2.550043;
   DATA[1291,1] := 796.7133;
   DATA[1291,2] := 2.0;
   DATA[1291,3] := 1.0;
   DATA[1291,4] := 262.5609;
   DATA[1291,5] := 8.464369;
   DATA[1291,6] := 317.6878;
   DATA[1291,8] := 1.0;
   DATA[1291,9] := 1.0;
   DATA[1291,10] := 1.0;
   DATA[1291,11] := 1.997567;
   DATA[1291,12] := 0.000256221;
   DATA[1291,13] := 1011.079;
   DATA[1291,14] := 1.0;
   DATA[1291,15] := 1.0;
   DATA[1291,16] := 1.0;
   DATA[1291,17] := 1.0;
   DATA[1291,18] := 1.0;
   DATA[1291,19] := 1.0;
   DATA[1291,20] := 148.808;
   DATA[1291,21] := 154.0118;
   DATA[1291,22] := 1.714798;
   DATA[1291,23] := 811.715;
   DATA[1291,24] := 2.0;
   DATA[1291,25] := 2.0;
   DATA[1291,26] := 7.87798;
   DATA[1291,27] := 143.0403;
   DATA[1291,28] := 263.0095;
   DATA[1291,29] := 12.26609;
   DATA[1291,30] := 1.723789;
   DATA[1291,31] := 1.289996;
   DATA[1291,32] := 0.7378293;
   DATA[1291,33] := 0.3082983;
   DATA[1291,34] := 2.0;
   DATA[1291,35] := 250.1762;
   DATA[1291,36] := 1.730048;
   DATA[1291,37] := 188.9419;
   DATA[1291,38] := 0.000128152;
   DATA[1291,39] := 1.0;
   DATA[1292,0] := 2.551965;
   DATA[1292,1] := 797.3412;
   DATA[1292,2] := 2.0;
   DATA[1292,3] := 1.0;
   DATA[1292,4] := 262.5609;
   DATA[1292,5] := 8.464369;
   DATA[1292,6] := 317.6878;
   DATA[1292,8] := 1.0;
   DATA[1292,9] := 1.0;
   DATA[1292,10] := 1.0;
   DATA[1292,11] := 1.997567;
   DATA[1292,12] := 0.000256221;
   DATA[1292,13] := 1011.52;
   DATA[1292,14] := 1.0;
   DATA[1292,15] := 1.0;
   DATA[1292,16] := 1.0;
   DATA[1292,17] := 1.0;
   DATA[1292,18] := 1.0;
   DATA[1292,19] := 1.0;
   DATA[1292,20] := 148.808;
   DATA[1292,21] := 154.0118;
   DATA[1292,22] := 1.714798;
   DATA[1292,23] := 811.5227;
   DATA[1292,24] := 2.0;
   DATA[1292,25] := 2.0;
   DATA[1292,26] := 7.87798;
   DATA[1292,27] := 143.0403;
   DATA[1292,28] := 263.0095;
   DATA[1292,29] := 12.26609;
   DATA[1292,30] := 1.723789;
   DATA[1292,31] := 1.290765;
   DATA[1292,32] := 0.7361649;
   DATA[1292,33] := 0.3082983;
   DATA[1292,34] := 2.0;
   DATA[1292,35] := 250.2403;
   DATA[1292,36] := 1.730048;
   DATA[1292,37] := 189.0861;
   DATA[1292,38] := 0.000128152;
   DATA[1292,39] := 1.0;
   DATA[1293,0] := 2.551965;
   DATA[1293,1] := 797.9693;
   DATA[1293,2] := 2.0;
   DATA[1293,3] := 1.0;
   DATA[1293,4] := 262.5609;
   DATA[1293,5] := 8.464369;
   DATA[1293,6] := 317.6878;
   DATA[1293,8] := 1.0;
   DATA[1293,9] := 1.0;
   DATA[1293,10] := 1.0;
   DATA[1293,11] := 1.997567;
   DATA[1293,12] := 0.000256221;
   DATA[1293,13] := 1010.919;
   DATA[1293,14] := 1.0;
   DATA[1293,15] := 1.0;
   DATA[1293,16] := 1.0;
   DATA[1293,17] := 1.0;
   DATA[1293,18] := 1.0;
   DATA[1293,19] := 1.0;
   DATA[1293,20] := 148.808;
   DATA[1293,21] := 153.8836;
   DATA[1293,22] := 1.714798;
   DATA[1293,23] := 811.4073;
   DATA[1293,24] := 2.0;
   DATA[1293,25] := 2.0;
   DATA[1293,26] := 7.87798;
   DATA[1293,27] := 143.0403;
   DATA[1293,28] := 263.0095;
   DATA[1293,29] := 12.26609;
   DATA[1293,30] := 1.724814;
   DATA[1293,31] := 1.282311;
   DATA[1293,32] := 0.7348846;
   DATA[1293,33] := 0.3082983;
   DATA[1293,34] := 2.0;
   DATA[1293,35] := 250.2403;
   DATA[1293,36] := 1.730048;
   DATA[1293,37] := 189.1342;
   DATA[1293,38] := 0.000128152;
   DATA[1293,39] := 1.0;
   DATA[1294,0] := 2.540115;
   DATA[1294,1] := 798.7544;
   DATA[1294,2] := 2.0;
   DATA[1294,3] := 1.0;
   DATA[1294,4] := 262.5609;
   DATA[1294,5] := 8.464369;
   DATA[1294,6] := 317.6878;
   DATA[1294,8] := 1.0;
   DATA[1294,9] := 1.0;
   DATA[1294,10] := 1.0;
   DATA[1294,11] := 1.997567;
   DATA[1294,12] := 0.000256221;
   DATA[1294,13] := 1011.039;
   DATA[1294,14] := 1.0;
   DATA[1294,15] := 1.0;
   DATA[1294,16] := 1.0;
   DATA[1294,17] := 1.0;
   DATA[1294,18] := 1.0;
   DATA[1294,19] := 1.0;
   DATA[1294,20] := 148.808;
   DATA[1294,21] := 153.8836;
   DATA[1294,22] := 1.714798;
   DATA[1294,23] := 810.9459;
   DATA[1294,24] := 2.0;
   DATA[1294,25] := 2.0;
   DATA[1294,26] := 7.87798;
   DATA[1294,27] := 143.0403;
   DATA[1294,28] := 263.0095;
   DATA[1294,29] := 11.88157;
   DATA[1294,30] := 1.726096;
   DATA[1294,31] := 1.27232;
   DATA[1294,32] := 0.7348846;
   DATA[1294,33] := 0.3082983;
   DATA[1294,34] := 2.0;
   DATA[1294,35] := 250.2403;
   DATA[1294,36] := 1.730048;
   DATA[1294,37] := 189.1342;
   DATA[1294,38] := 0.000128152;
   DATA[1294,39] := 1.0;
   DATA[1295,0] := 2.537232;
   DATA[1295,1] := 798.9506;
   DATA[1295,2] := 2.0;
   DATA[1295,3] := 1.0;
   DATA[1295,4] := 262.5609;
   DATA[1295,5] := 8.464369;
   DATA[1295,6] := 317.6878;
   DATA[1295,8] := 1.0;
   DATA[1295,9] := 1.0;
   DATA[1295,10] := 1.0;
   DATA[1295,11] := 1.997567;
   DATA[1295,12] := 0.000256221;
   DATA[1295,13] := 1010.718;
   DATA[1295,14] := 1.0;
   DATA[1295,15] := 1.0;
   DATA[1295,16] := 1.0;
   DATA[1295,17] := 1.0;
   DATA[1295,18] := 1.0;
   DATA[1295,19] := 1.0;
   DATA[1295,20] := 148.808;
   DATA[1295,21] := 153.8836;
   DATA[1295,22] := 1.715567;
   DATA[1295,23] := 810.8306;
   DATA[1295,24] := 2.0;
   DATA[1295,25] := 2.0;
   DATA[1295,26] := 7.87798;
   DATA[1295,27] := 143.0403;
   DATA[1295,28] := 263.0095;
   DATA[1295,29] := 11.88157;
   DATA[1295,30] := 1.726993;
   DATA[1295,31] := 1.271679;
   DATA[1295,32] := 0.7348846;
   DATA[1295,33] := 0.3082983;
   DATA[1295,34] := 2.0;
   DATA[1295,35] := 250.3525;
   DATA[1295,36] := 1.730048;
   DATA[1295,37] := 189.1342;
   DATA[1295,38] := 0.000128152;
   DATA[1295,39] := 1.0;
   DATA[1296,0] := 2.532428;
   DATA[1296,1] := 799.6179;
   DATA[1296,2] := 2.0;
   DATA[1296,3] := 1.0;
   DATA[1296,4] := 262.5609;
   DATA[1296,5] := 8.464369;
   DATA[1296,6] := 317.6878;
   DATA[1296,8] := 1.0;
   DATA[1296,9] := 1.0;
   DATA[1296,10] := 1.0;
   DATA[1296,11] := 1.997567;
   DATA[1296,12] := 0.000256221;
   DATA[1296,13] := 1011.079;
   DATA[1296,14] := 1.0;
   DATA[1296,15] := 1.0;
   DATA[1296,16] := 1.0;
   DATA[1296,17] := 1.0;
   DATA[1296,18] := 1.0;
   DATA[1296,19] := 1.0;
   DATA[1296,20] := 148.808;
   DATA[1296,21] := 153.8836;
   DATA[1296,22] := 1.716208;
   DATA[1296,23] := 810.1384;
